C01734=2169.363,-41.196,-377.460,-0.2119,7.1275,-90.0002
C01735=2166.065,-41.196,-377.214,1.4381,5.5003,-90.0002
C01736=2165.275,-41.196,-377.323,0.1088,3.4320,-90.0002
C01737=2163.485,-41.196,-377.080,0.8193,6.3311,-90.0002
C01738=2160.102,-41.196,-377.738,1.1974,2.9163,-90.0002
C01739=2158.853,-41.196,-377.593,-1.1287,2.0683,-90.0002
C01740=2155.073,-41.196,-378.064,1.3693,1.9251,-90.0002
C01741=2153.724,-41.196,-377.850,1.3521,2.0282,-90.0002
C01742=2150.349,-41.196,-378.400,0.7620,2.9793,-90.0002
C01743=2149.136,-41.196,-377.910,3.1168,3.6783,-90.0002
C01744=2145.160,-41.196,-378.700,1.6558,3.1684,-90.0002
C01745=2144.326,-41.196,-378.466,1.6902,3.9190,-90.0002
C01746=2140.135,-41.196,-378.318,-1.0255,1.1459,-90.0002
C01747=2138.981,-41.196,-379.103,0.0114,2.0683,-90.0002
C01748=2135.291,-41.196,-378.850,3.2715,3.0710,-90.0002
C01749=2133.841,-41.196,-379.406,0.1718,0.1776,-90.0002
C01750=2130.488,-41.196,-378.890,4.1482,2.5840,-90.0002
C01751=2128.923,-41.196,-379.018,1.7990,7.3567,-90.0002
C01752=2125.737,-41.196,-379.393,3.4893,0.4526,-90.0002
C01753=2123.975,-41.196,-378.591,2.5954,1.8391,-90.0002
C01754=2120.075,-41.196,-379.170,-0.6073,2.3090,-90.0002
C01755=2118.901,-41.196,-379.712,0.9167,4.8185,-90.0002
C01756=2114.735,-41.196,-380.002,-3.3174,-0.1260,-90.0002
C01757=2113.577,-41.196,-379.959,2.9621,-3.2601,-90.0002
C01758=2110.098,-41.196,-379.433,10.2272,3.8674,-90.0002
C01759=2109.561,-41.196,-379.487,3.1971,-2.4293,-90.0002
C01760=2105.376,-41.196,-380.509,4.7440,3.5007,-90.0002
C01761=2104.898,-41.196,-379.374,1.4438,2.9679,-90.0002
C01762=2100.737,-41.196,-379.764,1.3521,-0.0458,-90.0002
C01763=2099.790,-41.196,-380.834,-1.4725,0.2291,-90.0002
C01764=2095.224,-41.196,-380.131,4.6123,2.7501,-90.0002
C01765=2093.930,-41.196,-380.331,1.6042,7.5859,-90.0002
C01766=2089.893,-41.196,-380.417,3.3976,4.7612,-90.0002
C01767=2089.258,-41.196,-380.773,0.7792,-1.9251,-90.0002
C01768=2085.330,-41.196,-380.757,0.7906,0.8193,-90.0002
C01769=2083.879,-41.196,-379.511,3.0194,-1.3980,-90.0002
C01770=2079.836,-41.196,-380.416,0.6245,0.3151,-90.0002
C01771=2079.038,-41.196,-380.368,2.0569,-1.8793,-90.0002
C01772=2074.672,-41.196,-379.861,3.7987,2.4980,-90.0002
C01773=2074.092,-41.196,-380.658,7.0473,8.2448,-90.0002
C01774=2070.056,-41.196,-379.715,-0.4640,3.1569,-90.0002
C01775=2069.076,-41.196,-380.400,-0.3265,-1.2776,-90.0002
C01776=2065.277,-41.196,-380.250,-0.5672,3.2773,-90.0002
C01777=2063.880,-41.196,-379.731,2.2517,-1.3808,-90.0002
C01778=2060.201,-41.196,-379.972,1.1631,-1.2318,-90.0002
C01779=2059.099,-41.196,-380.740,8.2276,1.3808,-90.0002
C01780=2055.123,-41.196,-380.849,3.2887,0.3495,-90.0002
C01781=2053.996,-41.196,-380.050,6.7551,-2.2230,-90.0002
C01782=2049.819,-41.196,-380.443,5.9358,-0.0687,-90.0002
C01783=2049.134,-41.196,-381.700,0.0229,5.6608,-90.0002
C01784=2045.224,-41.196,-381.245,5.5233,1.9595,-90.0002
C01785=2044.771,-41.196,-380.905,-4.0278,-0.0744,-90.0002
C01786=2040.257,-41.196,-381.458,1.0943,4.4633,-90.0002
C01787=2039.336,-41.196,-379.745,0.8880,1.7532,-90.0002
C01788=2035.560,-41.196,-380.149,0.7276,-3.2372,-90.0002
C01789=2033.515,-41.196,-381.337,1.0141,-2.7731,-90.0002
C01790=2029.970,-41.196,-381.111,4.8758,2.0912,-90.0002
C01791=2028.017,-41.196,-380.702,0.7505,-0.9052,-90.0002
C01792=2025.281,-41.196,-380.401,5.3800,-0.4297,-90.0002
C01793=2023.851,-41.196,-380.213,0.4812,-2.4350,-90.0002
C01794=2019.728,-41.196,-380.300,2.4121,-2.4006,-90.0002
C01795=2019.058,-41.196,-381.536,1.7647,2.5954,-90.0002
C01796=2014.946,-41.196,-380.978,1.1860,-0.4870,-90.0002
C01797=2010.390,-41.196,-380.567,-1.6386,5.3342,-90.0002
C01798=2009.731,-41.196,-381.456,3.9648,1.5068,-90.0002
C01799=2006.217,-41.196,-381.020,0.1546,3.9935,-90.0002
C01800=2004.385,-41.196,-380.094,1.2204,2.7903,-90.0002
C01801=2001.248,-41.196,-381.863,6.6692,5.0821,-90.0002
C01802=2000.379,-41.196,-380.943,5.5863,0.5500,-90.0002
C01803=1997.761,-41.196,-382.132,2.2116,-0.1718,-90.0002
C01804=1995.113,-41.196,-381.971,0.2578,3.1054,-90.0002
C01805=1994.652,-41.196,-379.974,2.1886,1.7074,-90.0002
C01806=1989.787,-41.196,-381.076,2.2173,-1.1229,-90.0002
C01807=1989.016,-41.196,-379.930,2.3491,0.3896,-90.0002
C01808=1986.291,-41.196,-381.148,-1.1688,-0.7047,-90.0002
C01809=1984.627,-41.196,-380.667,5.7467,2.3433,-90.0002
C01810=1980.711,-41.196,-381.395,3.0939,-0.4812,-90.0002
C01811=1980.047,-41.196,-381.569,2.0168,-4.2799,-90.0002
C01812=1976.640,-41.196,-382.374,6.9728,-1.3407,-90.0002
C01813=1975.100,-41.196,-380.121,-2.7845,0.1375,-90.0002
C01814=1973.698,-41.196,-381.294,-0.0802,5.6092,-90.0002
C01815=1970.010,-41.196,-380.203,9.3162,-2.5152,-90.0002
C01816=1968.613,-41.196,-382.095,-1.0313,1.8449,-90.0002
C01817=1966.022,-41.196,-381.592,3.9992,2.5439,-90.0002
C01818=1964.655,-41.196,-380.029,2.1314,1.8391,-90.0002
C01819=1960.547,-41.196,-380.255,2.1657,1.7188,-90.0002
C01820=1959.422,-41.196,-380.031,8.5198,-1.8678,-90.0002
C01821=1957.473,-41.196,-382.205,3.0997,-0.7792,-90.0002
C01822=1955.043,-41.196,-381.735,4.3945,0.1375,-90.0002
C01823=1954.062,-41.196,-381.684,6.5546,1.5412,-90.0002
C01824=1950.141,-41.196,-380.586,4.7956,0.8250,-90.0002
C01825=1949.476,-41.196,-381.977,1.8162,-8.2334,-90.0002
C01826=1945.507,-41.196,-381.667,1.2776,5.7926,-90.0002
C01827=1944.984,-41.196,-381.700,3.3861,2.4121,-90.0002
C01828=1943.695,-41.196,-382.237,-0.0114,2.3777,-90.0002
C01829=1941.079,-41.196,-381.081,1.8048,4.4633,-90.0002
C01830=1939.451,-41.196,-380.357,0.5385,3.7815,-90.0002
C01831=1935.406,-41.196,-381.487,2.2288,-1.6902,-90.0002
C01832=1934.176,-41.196,-380.632,5.7467,-0.7620,-90.0002
C01833=1930.488,-41.196,-381.185,6.1592,-2.4178,-90.0002
C01834=1929.880,-41.196,-381.659,-1.6844,0.4927,-90.0002
C01835=1926.074,-41.196,-380.394,0.8422,4.2112,-90.0002
C01836=1924.491,-41.196,-380.870,6.9728,-0.0974,-90.0002
C01837=1920.888,-41.196,-380.599,4.3201,4.1482,-90.0002
C01838=1920.372,-41.196,-381.287,7.0588,-6.8583,-90.0002
C01839=1919.171,-41.196,-382.295,0.0057,2.4465,-90.0002
C01840=1915.534,-41.196,-381.857,-6.9958,13.2295,-90.0002
C01841=1914.581,-41.196,-381.964,10.5137,-7.5401,-90.0002
C01842=1910.831,-41.196,-382.252,3.8846,-4.1825,-90.0002
C01843=1909.397,-41.196,-381.109,5.8040,0.4411,-90.0002
C01844=1905.433,-41.196,-381.982,5.2654,-2.9220,-90.0002
C01845=1904.354,-41.196,-380.850,4.1539,-1.1573,-90.0002
C01846=1901.224,-41.196,-380.146,1.1917,2.7845,-90.0002
C01847=1900.943,-41.196,-382.312,1.3407,-1.5813,-90.0002
C01848=1898.677,-41.196,-381.742,-0.9224,1.3235,-90.0002
C01849=1895.878,-41.196,-381.910,3.6096,-0.0630,-90.0002
C01850=1895.638,-41.196,-380.243,2.0397,1.5412,-90.0002
C01851=1892.807,-41.196,-382.261,0.9625,0.2005,-90.0002
C01852=1890.565,-41.196,-380.594,1.7074,1.1573,-90.0002
C01853=1889.860,-41.196,-381.233,-0.7964,-1.0599,-90.0002
C01854=1885.286,-41.196,-382.385,0.5786,1.4266,-90.0002
C01855=1884.612,-41.196,-380.791,1.2948,-0.9453,-90.0002
C01856=1882.779,-41.196,-382.009,3.6841,1.0370,-90.0002
C01857=1880.149,-41.196,-381.749,2.3720,-5.9301,-90.0002
C01858=1878.438,-41.196,-380.761,0.9511,-0.3609,-90.0002
C01859=1875.006,-41.196,-382.215,1.3063,-5.0935,-90.0002
C01860=1874.154,-41.196,-381.613,-1.0599,-0.8594,-90.0002
C01861=1870.916,-41.196,-381.373,1.7704,3.4893,-90.0002
C01862=1869.849,-41.196,-381.316,-0.6531,0.3896,-90.0002
C01863=1866.246,-41.196,-382.056,-1.6844,-6.2223,-90.0002
C01864=1864.858,-41.196,-379.990,2.8246,1.7761,-90.0002
C01865=1864.164,-41.196,-381.007,3.0022,0.7677,-90.0002
C01866=1859.806,-41.196,-380.511,1.6100,0.7677,-90.0002
C01867=1859.069,-41.196,-381.389,0.2521,-0.2922,-90.0002
C01868=1854.817,-41.196,-379.850,0.1489,4.6123,-90.0002
C01869=1853.868,-41.196,-381.034,5.8900,-1.4323,-90.0002
C01870=1850.003,-41.196,-380.905,2.6470,-0.5156,-90.0002
C01871=1848.676,-41.196,-380.548,0.7734,1.9938,-90.0002
C01872=1844.734,-41.196,-380.810,-1.4209,0.5958,-90.0002
C01873=1844.143,-41.196,-380.694,-1.6501,-0.9854,-90.0002
C01874=1840.047,-41.196,-379.707,4.4518,-5.9473,-90.0002
C01875=1838.314,-41.196,-379.343,1.3636,-3.0252,-90.0002
C01876=1834.393,-41.196,-379.620,-2.1084,0.3380,-90.0002
C01877=1833.918,-41.196,-380.668,2.2746,-6.1936,-90.0002
C01878=1829.774,-41.196,-379.832,-0.7448,-2.4522,-90.0002
C01879=1825.669,-41.196,-379.624,6.4973,-3.8903,-90.0002
C01880=1825.187,-41.196,-379.253,3.0825,-5.2368,-90.0002
C01881=1820.708,-41.196,-378.938,2.6871,-3.0137,-90.0002
C01882=1819.044,-41.196,-379.962,-0.4469,1.3120,-90.0002
C01883=1815.594,-41.196,-379.344,3.0194,-0.9224,-90.0002
C01884=1814.615,-41.196,-378.950,3.4320,-2.8132,-90.0002
C01885=1810.688,-41.196,-379.312,-0.1661,-2.1027,-90.0002
C01886=1809.855,-41.196,-379.145,4.2857,-2.7673,-90.0002
C01887=1805.671,-41.196,-378.925,0.2922,-3.3747,-90.0002
C01888=1804.704,-41.196,-378.996,2.3605,-4.5492,-90.0002
C01889=1800.366,-41.196,-378.306,4.3201,-5.8327,-90.0002
C01890=1799.418,-41.196,-378.526,-5.2941,-12.6394,-90.0002
C01891=1795.305,-91.196,-377.541,1.0542,7.1104,-90.0002
C01892=1799.418,-91.196,-377.424,1.8162,-5.2712,-90.0002
C01893=1800.080,-91.196,-377.530,-0.8995,-6.1134,-90.0002
C01894=1804.178,-91.196,-377.422,0.5271,-1.1631,-90.0002
C01895=1805.558,-91.196,-378.041,2.7272,-4.0794,-90.0002
C01896=1809.552,-91.196,-378.343,-0.9224,3.0997,-90.0002
C01897=1810.802,-91.196,-377.922,2.2803,-1.4037,-90.0002
C01898=1814.674,-91.196,-377.946,-0.2177,2.1543,-90.0002
C01899=1816.221,-91.196,-377.447,4.0278,1.1401,-90.0002
C01900=1819.459,-91.196,-378.316,0.6245,-1.4495,-90.0002
C01901=1820.188,-91.196,-378.633,3.9190,-3.7757,-90.0002
C01902=1823.981,-91.196,-378.201,0.4984,0.5786,-90.0002
C01903=1825.225,-91.196,-377.414,3.6039,0.5729,-90.0002
C01904=1829.473,-91.196,-377.953,3.6898,0.2119,-90.0002
C01905=1830.985,-91.196,-378.696,-0.7906,0.8307,-90.0002
C01906=1834.377,-91.196,-377.651,1.8506,3.2544,-90.0002
C01907=1835.959,-91.196,-377.260,0.4640,-0.9568,-90.0002
C01908=1839.694,-91.196,-377.295,2.4923,-0.5213,-90.0002
C01909=1840.541,-91.196,-378.454,2.9507,-6.2395,-90.0002
C01910=1844.696,-91.196,-377.160,0.1948,2.4064,-90.0002
C01911=1845.955,-91.196,-377.972,3.5809,-0.0744,-90.0002
C01912=1848.927,-91.196,-378.948,6.5145,-2.1428,-90.0002
C01913=1849.965,-91.196,-377.457,4.4518,1.1516,-90.0002
C01914=1851.787,-91.196,-376.910,4.3258,-2.3949,-90.0002
C01915=1854.842,-91.196,-377.542,1.1401,2.7501,-90.0002
C01916=1855.268,-91.196,-378.573,2.6699,-0.3781,-90.0002
C01917=1859.702,-91.196,-378.097,3.0481,0.3781,-90.0002
C01918=1860.339,-91.196,-377.126,1.4839,4.8930,-90.0002
C01919=1864.837,-91.196,-377.522,2.1600,-1.5870,-90.0002
C01920=1866.502,-91.196,-378.692,-1.9938,1.4323,-90.0002
C01921=1869.655,-91.196,-379.088,5.2712,0.2807,-90.0002
C01922=1870.902,-91.196,-378.347,3.7929,3.7471,-90.0002
C01923=1874.608,-91.196,-378.370,7.1275,-2.7215,-90.0002
C01924=1875.701,-91.196,-377.271,2.4694,1.8964,-90.0002
C01925=1879.089,-91.196,-376.878,2.4522,0.1890,-90.0002
C01926=1880.404,-91.196,-377.206,2.2918,-0.0229,-90.0002
C01927=1883.226,-91.196,-379.326,1.9767,-3.0366,-90.0002
C01928=1884.972,-91.196,-378.617,0.3953,1.4094,-90.0002
C01929=1889.337,-91.196,-377.344,5.2597,-0.7391,-90.0002
C01930=1890.538,-91.196,-377.879,3.6726,0.8880,-90.0002
C01931=1894.036,-91.196,-376.879,1.2948,2.3605,-90.0002
C01932=1895.783,-91.196,-378.730,7.9984,-2.5496,-90.0002
C01933=1899.291,-91.196,-379.024,3.5179,0.5156,-90.0002
C01934=1900.259,-91.196,-378.071,3.0022,-0.2807,-90.0002
C01935=1902.386,-91.196,-377.434,4.2341,-4.2742,-90.0002
C01936=1905.020,-91.196,-378.297,11.6596,4.2055,-90.0002
C01937=1907.374,-91.196,-379.871,1.9652,2.2459,-90.0002
C01938=1909.572,-91.196,-377.869,1.4839,1.8964,-90.0002
C01939=1910.710,-91.196,-377.032,4.0508,-1.7589,-90.0002
C01940=1914.960,-91.196,-379.427,4.7841,0.5786,-90.0002
C01941=1915.743,-91.196,-378.526,1.3235,-1.5297,-90.0002
C01942=1920.119,-91.196,-379.065,4.4919,1.5297,-90.0002
C01943=1920.959,-91.196,-378.296,-0.0229,4.7612,-90.0002
C01944=1924.741,-91.196,-380.206,2.2402,0.7563,-90.0002
C01945=1925.292,-91.196,-378.183,2.6757,-5.1050,-90.0002
C01946=1930.023,-91.196,-377.070,6.5202,3.2715,-90.0002
C01947=1930.189,-91.196,-378.390,5.8842,1.1287,-90.0002
C01948=1934.079,-91.196,-376.687,-2.3835,0.8365,-90.0002
C01949=1935.446,-91.196,-379.999,3.5065,1.0828,-90.0002
C01950=1938.838,-91.196,-377.816,2.6356,-0.9682,-90.0002
C01951=1940.436,-91.196,-378.391,4.4346,1.6157,-90.0002
C01952=1942.886,-91.196,-379.959,0.6932,2.2116,-90.0002
C01953=1944.917,-91.196,-377.943,4.2799,1.9365,-90.0002
C01954=1948.261,-91.196,-377.396,3.0595,1.5469,-90.0002
C01955=1949.956,-91.196,-378.329,1.3349,0.4984,-90.0002
C01956=1953.464,-91.196,-377.372,3.5179,-1.6730,-90.0002
C01957=1955.037,-91.196,-379.269,1.9365,2.7960,-90.0002
C01958=1957.644,-91.196,-377.607,1.7475,2.2689,-90.0002
C01959=1959.560,-91.196,-379.741,2.5783,7.5802,-90.0002
C01960=1963.395,-91.196,-378.215,7.7463,0.4411,-90.0002
C01961=1964.946,-91.196,-376.641,3.7643,-0.8537,-90.0002
C01962=1969.099,-91.196,-378.729,5.1050,1.8506,-90.0002
C01963=1970.306,-91.196,-377.055,3.7414,-0.1833,-90.0002
C01964=1972.157,-91.196,-376.780,0.7792,1.5584,-90.0002
C01965=1974.946,-91.196,-378.646,2.7158,-0.2692,-90.0002
C01966=1975.717,-91.196,-379.977,7.0359,0.8766,-90.0002
C01967=1979.866,-91.196,-378.788,-0.4755,-0.8250,-90.0002
C01968=1981.044,-91.196,-377.480,2.2918,0.4640,-90.0002
C01969=1984.927,-91.196,-379.068,4.5607,0.6589,-90.0002
C01970=1987.335,-91.196,-376.378,4.2055,2.3491,-90.0002
C01971=1990.373,-91.196,-378.245,3.0080,1.4266,-90.0002
C01972=1992.305,-91.196,-379.490,2.4236,0.7964,-90.0002
C01973=1994.371,-91.196,-379.740,6.0790,0.5500,-90.0002
C01974=1995.503,-91.196,-379.443,0.4927,-1.7761,-90.0002
C01975=1999.561,-91.196,-377.473,1.5183,2.2173,-90.0002
C01976=2000.080,-91.196,-379.228,1.2891,2.9621,-90.0002
C01977=2004.406,-91.196,-378.900,-1.6501,2.0683,-90.0002
C01978=2005.652,-91.196,-377.941,2.6184,0.8021,-90.0002
C01979=2009.434,-91.196,-378.794,0.4239,-3.4492,-90.0002
C01980=2010.261,-91.196,-377.289,2.8361,-0.6245,-90.0002
C01981=2013.853,-91.196,-379.442,2.9621,4.2112,-90.0002
C01982=2015.071,-91.196,-377.219,2.6585,2.2402,-90.0002
C01983=2019.320,-91.196,-379.177,3.7815,-0.5844,-90.0002
C01984=2020.278,-91.196,-377.598,4.4919,3.1226,-90.0002
C01985=2024.061,-91.196,-378.312,1.9365,2.6012,-90.0002
C01986=2024.673,-91.196,-377.500,5.7467,1.0485,-90.0002
C01987=2028.765,-91.196,-377.287,3.8388,-5.4717,-90.0002
C01988=2029.403,-91.196,-379.302,-2.2345,-1.3063,-90.0002
C01989=2033.995,-91.196,-379.271,2.9278,1.7246,-90.0002
C01990=2035.196,-91.196,-377.121,4.8185,0.4526,-90.0002
C01991=2036.257,-91.196,-376.721,10.1528,2.3720,-90.0002
C01992=2040.109,-91.196,-378.754,7.9354,0.5500,-90.0002
C01993=2041.225,-91.196,-377.911,-0.4411,1.0657,-90.0002
C01994=2044.180,-91.196,-379.373,2.9335,-1.6386,-90.0002
C01995=2044.990,-91.196,-377.271,1.3521,4.0164,-90.0002
C01996=2049.316,-91.196,-379.066,6.3025,-1.2662,-90.0002
C01997=2050.431,-91.196,-379.407,0.5786,1.3865,-90.0002
C01998=2054.812,-91.196,-378.624,0.2234,0.9625,-90.0002
C01999=2055.478,-91.196,-377.232,6.3999,-2.6356,-90.0002
C02000=2059.087,-91.196,-379.472,4.1825,1.1229,-90.0002
C02001=2060.348,-91.196,-379.251,4.4862,4.9045,-90.0002
C02002=2064.525,-91.196,-377.693,3.4320,0.2521,-90.0002
C02003=2065.787,-91.196,-377.027,1.9308,-1.4725,-90.0002
C02004=2067.675,-91.196,-377.871,5.0305,-0.0630,-90.0002
C02005=2069.595,-91.196,-376.894,2.4694,1.2433,-90.0002
C02006=2070.674,-91.196,-378.584,6.5947,2.0053,-90.0002
C02007=2074.375,-91.196,-378.345,4.0393,-0.8021,-90.0002
C02008=2075.996,-91.196,-378.574,2.9564,-0.6359,-90.0002
C02009=2079.628,-91.196,-379.307,-2.1314,-1.5183,-90.0002
C02010=2080.836,-91.196,-378.302,5.6837,1.9079,-90.0002
C02011=2084.764,-91.196,-378.169,-0.6932,0.1145,-90.0002
C02012=2086.437,-91.196,-376.636,5.5977,-1.2032,-90.0002
C02013=2089.410,-91.196,-378.030,0.8766,3.1569,-90.0002
C02014=2090.183,-91.196,-377.411,2.8647,3.1111,-90.0002
C02015=2094.448,-91.196,-378.114,2.3032,-0.5901,-90.0002
C02016=2096.058,-91.196,-377.332,1.9767,2.8590,-90.0002
C02017=2099.543,-91.196,-377.890,6.0160,0.3380,-90.0002
C02018=2100.315,-91.196,-378.222,3.9534,-0.4297,-90.0002
C02019=2104.184,-91.196,-376.632,5.2024,-2.3777,-90.0002
C02020=2104.790,-91.196,-377.159,2.6642,0.0802,-90.0002
C02021=2107.833,-91.196,-376.917,4.3544,1.6673,-90.0002
C02022=2110.286,-91.196,-378.242,5.9301,1.0599,-90.0002
C02023=2111.691,-91.196,-377.226,4.3659,6.2108,-90.0002
C02024=2114.634,-91.196,-378.486,0.7964,-1.5527,-90.0002
C02025=2116.213,-91.196,-378.735,6.7150,2.4579,-90.0002
C02026=2119.530,-91.196,-376.715,0.9453,-0.0572,-90.0002
C02027=2121.044,-91.196,-377.621,1.9136,2.3090,-90.0002
C02028=2124.313,-91.196,-377.459,4.4633,4.2456,-90.0002
C02029=2125.062,-91.196,-377.243,4.1711,-1.2891,-90.0002
C02030=2128.421,-91.196,-376.976,5.2425,3.3575,-90.0002
C02031=2129.559,-91.196,-377.491,1.8277,3.9476,-90.0002
C02032=2131.041,-91.196,-378.289,2.2975,4.6581,-90.0002
C02033=2134.586,-91.196,-377.315,2.7731,2.5095,-90.0002
C02034=2135.602,-91.196,-377.583,1.8162,2.5382,-90.0002
C02035=2138.526,-91.196,-377.954,1.0084,4.3029,-90.0002
C02036=2140.068,-91.196,-376.562,2.3032,4.4919,-90.0002
C02037=2141.212,-91.196,-376.416,1.2032,6.1478,-90.0002
C02038=2144.686,-91.196,-376.860,0.7448,1.8964,-90.0002
C02039=2145.499,-91.196,-376.622,1.1344,0.4239,-90.0002
C02040=2149.245,-91.196,-377.512,3.1512,1.4209,-90.0002
C02041=2150.530,-91.196,-376.290,2.6871,1.9652,-90.0002
C02042=2154.261,-91.196,-375.625,1.7818,4.1711,-90.0002
C02043=2155.389,-91.196,-377.406,-0.5328,5.5003,-90.0002
C02044=2158.923,-91.196,-376.796,3.0424,2.1027,-90.0002
C02045=2159.995,-91.196,-377.108,2.1886,5.3800,-90.0002
C02046=2162.658,-91.196,-377.093,-2.9278,1.2776,-90.0002
C02047=2165.115,-91.196,-376.774,-1.1459,1.9767,-90.0002
C02048=2166.465,-91.196,-376.259,1.1344,0.3208,-90.0002
C02049=2169.854,-91.196,-376.573,2.2631,3.6096,-90.0002
C02050=2171.046,-91.196,-376.056,-0.4526,0.4812,-90.0002
C02051=2174.160,-91.196,-376.291,4.0278,3.7987,-90.0002
C02052=2175.265,-91.196,-375.729,4.2398,3.4434,-90.0002
C02053=2179.561,-91.196,-375.441,-1.2948,4.6810,-90.0002
C02054=2180.555,-91.196,-376.351,3.7184,6.6978,-90.0002
C02055=2184.038,-91.196,-375.049,-0.9453,5.4201,-90.0002
C02056=2185.498,-91.196,-374.824,6.5374,3.6268,-90.0002
C02057=2185.415,-141.196,-374.060,2.6699,2.4178,-90.0002
C02058=2184.214,-141.196,-373.905,3.8388,-0.5328,-90.0002
C02059=2180.012,-141.196,-374.573,-0.2750,1.7188,-90.0002
C02060=2179.127,-141.196,-373.260,4.8414,1.6558,-90.0002
C02061=2175.684,-141.196,-373.842,2.8074,1.6157,-90.0002
C02062=2174.219,-141.196,-375.290,0.1203,1.9938,-90.0002
C02063=2170.489,-141.196,-374.723,0.7505,-0.1432,-90.0002
C02064=2169.134,-141.196,-375.269,2.4465,0.8823,-90.0002
C02065=2165.315,-141.196,-373.747,5.3399,2.9450,-90.0002
C02066=2164.630,-141.196,-375.232,1.5928,-2.0511,-90.0002
C02067=2160.260,-141.196,-374.253,3.2486,-0.4755,-90.0002
C02068=2159.387,-141.196,-375.240,3.2085,2.3204,-90.0002
C02069=2155.362,-141.196,-374.889,3.2601,2.3376,-90.0002
C02070=2154.922,-141.196,-375.396,1.6443,-3.1054,-90.0002
C02071=2150.433,-141.196,-374.026,6.6119,0.3208,-90.0002
C02072=2149.135,-141.196,-374.393,2.4350,0.5901,-90.0002
C02073=2145.477,-141.196,-375.714,3.7356,1.0370,-90.0002
C02074=2144.146,-141.196,-373.491,9.5512,2.5897,-90.0002
C02075=2140.769,-141.196,-374.776,5.0248,-0.2922,-90.0002
C02076=2139.289,-141.196,-373.542,7.4140,-1.3922,-90.0002
C02077=2135.263,-141.196,-375.429,7.3510,0.1833,-90.0002
C02078=2133.968,-141.196,-373.056,1.0886,0.0744,-90.0002
C02079=2130.077,-141.196,-375.677,3.5408,2.3204,-90.0002
C02080=2129.113,-141.196,-373.373,6.1077,-0.3609,-90.0002
C02081=2125.272,-141.196,-375.578,2.2345,-0.4755,-90.0002
C02082=2124.761,-141.196,-376.048,2.3835,1.5240,-90.0002
C02083=2120.328,-141.196,-375.059,4.2799,3.1856,-90.0002
C02084=2118.606,-141.196,-375.500,2.9048,-1.3407,-90.0002
C02085=2115.318,-141.196,-372.750,6.7666,5.3055,-90.0002
C02086=2113.745,-141.196,-375.727,1.9423,2.2116,-90.0002
C02087=2110.355,-141.196,-376.311,2.8762,2.6642,-90.0002
C02088=2109.416,-141.196,-375.774,2.6757,1.2146,-90.0002
C02089=2105.001,-141.196,-375.638,5.5061,-0.5557,-90.0002
C02090=2104.265,-141.196,-372.948,9.5397,-1.5412,-90.0002
C02091=2100.516,-141.196,-375.890,3.7815,0.3208,-90.0002
C02092=2099.725,-141.196,-375.017,5.3514,2.5954,-90.0002
C02093=2095.436,-141.196,-374.505,3.1340,-2.1886,-90.0002
C02094=2094.167,-141.196,-374.712,7.3968,-1.4725,-90.0002
C02095=2090.205,-141.196,-375.986,1.2204,-0.8938,-90.0002
C02096=2089.109,-141.196,-374.205,4.1310,-2.1715,-90.0002
C02097=2085.580,-141.196,-375.997,3.4148,-0.6703,-90.0002
C02098=2084.360,-141.196,-374.346,4.7727,-0.3495,-90.0002
C02099=2080.253,-141.196,-373.722,6.0160,1.6902,-90.0002
C02100=2079.835,-141.196,-376.286,5.4602,1.1000,-90.0002
C02101=2074.913,-141.196,-376.787,5.9702,-1.1172,-90.0002
C02102=2073.522,-141.196,-375.699,5.3055,-0.2922,-90.0002
C02103=2069.173,-141.196,-373.234,4.2226,0.9281,-90.0002
C02104=2066.401,-141.196,-374.355,0.6760,1.9365,-90.0002
C02105=2064.927,-141.196,-375.525,1.1631,1.4495,-90.0002
C02106=2061.460,-141.196,-375.886,-0.9912,3.4033,-90.0002
C02107=2059.609,-141.196,-376.501,3.9648,-1.4495,-90.0002
C02108=2055.666,-141.196,-376.502,3.8903,0.3380,-90.0002
C02109=2055.045,-141.196,-375.888,1.5641,-0.8307,-90.0002
C02110=2051.232,-141.196,-374.111,-0.0171,1.5297,-90.0002
C02111=2049.797,-141.196,-376.208,7.0989,1.1287,-90.0002
C02112=2046.719,-141.196,-376.168,5.1508,1.7131,-90.0002
C02113=2045.239,-141.196,-372.335,-0.4927,-0.3609,-90.0002
C02114=2041.406,-141.196,-374.903,1.2433,1.2032,-90.0002
C02115=2039.762,-141.196,-374.660,3.5007,0.2291,-90.0002
C02116=2036.008,-141.196,-373.939,10.2158,2.8017,-90.0002
C02117=2034.926,-141.196,-373.407,8.3823,-1.5756,-90.0002
C02118=2030.385,-141.196,-374.996,4.5951,-1.0198,-90.0002
C02119=2029.826,-141.196,-374.272,9.8319,-2.3204,-90.0002
C02120=2026.054,-141.196,-375.886,3.5351,0.4812,-90.0002
C02121=2024.793,-141.196,-372.708,0.9339,2.4236,-90.0002
C02122=2020.791,-141.196,-373.674,11.6997,-2.9450,-90.0002
C02123=2019.172,-141.196,-375.199,3.9133,-0.1948,-90.0002
C02124=2016.262,-141.196,-377.076,2.7845,5.8728,-90.0002
C02125=2014.369,-141.196,-375.197,2.3720,0.4239,-90.0002
C02126=2010.352,-141.196,-374.971,4.6810,0.2864,-90.0002
C02127=2009.288,-141.196,-376.093,6.0504,0.8594,-90.0002
C02128=2005.597,-141.196,-375.731,5.6780,0.0802,-90.0002
C02129=2004.514,-141.196,-376.381,6.5890,-0.5786,-90.0002
C02130=2000.011,-141.196,-373.316,8.7719,4.5034,-90.0002
C02131=1998.643,-141.196,-376.369,3.5637,-1.1229,-90.0002
C02132=1995.495,-141.196,-375.756,6.1478,4.0966,-90.0002
C02133=1994.531,-141.196,-374.155,9.4251,-1.5011,-90.0002
C02134=1990.070,-141.196,-375.098,3.0653,-0.6646,-90.0002
C02135=1989.589,-141.196,-374.441,5.6608,3.1111,-90.0002
C02136=1984.910,-141.196,-374.777,0.8078,4.3716,-90.0002
C02137=1983.861,-141.196,-374.952,4.2971,3.1398,-90.0002
C02138=1980.391,-141.196,-374.252,6.0561,0.0744,-90.0002
C02139=1979.309,-141.196,-375.340,3.8617,1.5641,-90.0002
C02140=1975.109,-141.196,-376.260,6.2051,1.6214,-90.0002
C02141=1974.206,-141.196,-375.762,3.0538,0.6302,-90.0002
C02142=1970.228,-141.196,-374.936,2.1428,1.0599,-90.0002
C02143=1969.207,-141.196,-375.892,6.8697,0.3265,-90.0002
C02144=1965.515,-141.196,-375.103,3.5924,-0.9682,-90.0002
C02145=1964.102,-141.196,-376.394,5.5691,-2.4809,-90.0002
C02146=1959.717,-141.196,-375.815,4.2513,-0.8537,-90.0002
C02147=1959.054,-141.196,-373.895,3.7184,3.0767,-90.0002
C02148=1954.785,-141.196,-374.983,3.5236,0.0859,-90.0002
C02149=1954.384,-141.196,-375.969,-0.4239,3.3632,-97.1679
C02150=1950.054,-141.196,-375.487,2.4293,0.0458,-90.0002
C02151=1949.440,-141.196,-375.245,4.0565,-0.9110,-90.0002
C02152=1945.526,-141.196,-376.724,4.3602,-2.4522,-90.0002
C02153=1944.222,-141.196,-374.130,9.6027,-4.0107,-90.0002
C02154=1940.229,-141.196,-376.375,5.8842,1.6902,-90.0002
C02155=1939.527,-141.196,-377.085,-0.1088,1.1287,-90.0002
C02156=1935.213,-141.196,-373.944,3.5867,-1.9652,-90.0002
C02157=1934.819,-141.196,-375.337,5.0133,1.1058,-90.0002
C02158=1930.636,-141.196,-375.890,2.6012,0.0401,-90.0002
C02159=1929.735,-141.196,-376.410,1.7360,0.2005,-90.0002
C02160=1925.900,-141.196,-375.823,4.8987,-0.6646,-90.0002
C02161=1924.700,-141.196,-373.832,4.6696,-0.6818,-90.0002
C02162=1920.470,-141.196,-376.522,1.8964,1.4839,-90.0002
C02163=1919.832,-141.196,-376.398,7.0588,-1.1631,-90.0002
C02164=1916.892,-141.196,-375.801,5.0305,0.0802,-90.0002
C02165=1915.052,-141.196,-373.246,1.3750,1.9423,-90.0002
C02166=1912.060,-141.196,-376.956,4.9790,-0.6302,-90.0002
C02167=1910.298,-141.196,-375.968,2.0511,1.5412,-90.0002
C02168=1908.582,-141.196,-376.159,2.2975,3.9190,-90.0002
C02169=1905.388,-141.196,-373.909,6.9098,-4.0336,-90.0002
C02170=1903.985,-141.196,-376.680,3.2314,-0.8250,-90.0002
C02171=1900.049,-141.196,-376.768,-0.3093,0.4068,-90.0002
C02172=1899.194,-141.196,-376.566,4.7383,2.8819,-90.0002
C02173=1895.499,-141.196,-374.703,3.2715,2.5954,-90.0002
C02174=1894.268,-141.196,-376.976,1.5240,-1.5355,-90.0002
C02175=1890.500,-141.196,-375.186,9.5913,3.0080,-90.0002
C02176=1889.495,-141.196,-376.046,3.0080,0.1031,-90.0002
C02177=1885.342,-141.196,-376.640,3.3976,-0.3495,-90.0002
C02178=1885.135,-141.196,-375.791,3.1512,-0.9167,-90.0002
C02179=1879.748,-141.196,-375.833,6.2509,-0.8880,-90.0002
C02180=1878.976,-141.196,-375.179,7.6088,-2.4236,-90.0002
C02181=1875.506,-141.196,-376.619,9.7116,-2.7330,-90.0002
C02182=1874.493,-141.196,-374.949,6.0504,0.3609,-90.0002
C02183=1870.194,-141.196,-374.646,5.2540,3.8617,-90.0002
C02184=1869.293,-141.196,-375.463,3.0366,-0.4984,-90.0002
C02185=1865.075,-141.196,-376.316,2.4064,1.6787,-90.0002
C02186=1864.404,-141.196,-375.624,0.4125,2.3376,-90.0002
C02187=1859.803,-141.196,-375.872,2.1715,0.4927,-90.0002
C02188=1858.398,-141.196,-375.605,3.1340,-0.1432,-90.0002
C02189=1854.864,-141.196,-375.996,3.0767,-0.0859,-90.0002
C02190=1853.834,-141.196,-374.837,2.2918,1.4266,-90.0002
C02191=1850.410,-141.196,-375.284,2.2746,3.0080,-90.0002
C02192=1849.748,-141.196,-375.547,2.7501,1.1172,-90.0002
C02193=1845.055,-141.196,-375.674,3.4090,5.7123,-90.0002
C02194=1844.434,-141.196,-377.106,-3.7643,7.5401,-90.0002
C02195=1840.894,-141.196,-375.702,1.3063,-0.7333,-90.0002
C02196=1839.805,-141.196,-376.567,1.8621,1.5813,-90.0002
C02197=1835.935,-141.196,-377.111,1.0198,-2.9908,-90.0002
C02198=1834.687,-141.196,-375.834,8.2964,1.2547,-90.0002
C02199=1832.895,-141.196,-376.758,1.9022,-0.5213,-90.0002
C02200=1829.331,-141.196,-375.944,13.2410,2.8304,-90.0002
C02201=1825.616,-141.196,-376.772,2.5496,-2.2975,-90.0002
C02202=1824.719,-141.196,-376.707,-0.7161,2.4236,-90.0002
C02203=1823.375,-141.196,-376.275,1.4610,2.5954,-90.0002
C02204=1820.148,-141.196,-376.699,0.9224,1.9022,-90.0002
C02205=1819.386,-141.196,-377.239,-0.7333,7.9411,-90.0002
C02206=1817.633,-141.196,-377.017,-4.0794,7.6203,-90.0002
C02207=1815.194,-141.196,-377.208,0.9224,0.3208,-90.0002
C02208=1813.793,-141.196,-377.163,2.0741,-0.5271,-90.0002
C02209=1810.514,-141.196,-376.879,1.0370,0.4583,-90.0002
C02210=1809.304,-141.196,-376.514,5.6035,5.9358,-90.0002
C02211=1805.917,-141.196,-377.286,1.4438,1.7016,-90.0002
C02212=1805.150,-141.196,-377.071,-1.3120,3.1398,-90.0002
C02213=1803.613,-141.196,-376.936,4.8357,-1.0198,-90.0002
C02214=1800.646,-141.196,-376.815,1.7417,1.7475,-90.0002
C02215=1799.896,-141.196,-377.079,-1.0026,0.1203,-90.0002
C02216=1798.042,-141.196,-377.026,0.1088,5.4488,-90.0002
C02217=1794.253,-141.196,-377.324,1.7188,11.2528,-90.0002
C02218=1812.109,341.105,-503.612,89.8111,-0.2349,0.0000
C02219=2127.650,341.132,-503.612,90.5788,-0.2750,0.0000
C02220=2159.023,341.159,-503.612,90.6075,-0.4927,-0.0057
C02221=1816.234,341.190,-503.612,89.6048,0.1546,0.0000
C02222=1821.738,341.222,-503.612,90.0002,0.0687,0.0000
C02223=1812.786,341.237,-503.612,89.4559,-0.2922,0.0000
C02224=1809.568,341.249,-503.612,83.1648,0.5213,-0.0630
C02225=1831.712,341.267,-503.612,89.6621,0.4927,-0.0057
C02226=1826.384,341.287,-503.612,89.5475,0.2119,0.0000
C02227=1835.441,341.299,-503.612,89.7309,0.1145,0.0000
C02228=1840.177,341.323,-503.612,89.6736,0.4583,0.0000
C02229=1835.884,341.334,-503.612,89.8798,0.2406,0.0000
C02230=2119.313,341.341,-503.612,89.6335,0.1489,0.0000
C02231=2152.042,341.346,-503.612,90.8309,0.0229,0.0000
C02232=2175.237,341.354,-503.612,90.0403,0.4068,0.0000
C02233=1808.484,341.385,-503.612,89.6163,-1.0026,0.0057
C02234=2144.675,341.398,-503.612,90.8596,-0.2807,-0.0057
C02235=1798.586,341.407,-503.612,89.6392,0.8365,-0.0057
C02236=1838.296,341.417,-503.612,89.5361,-0.7677,0.0057
C02237=2112.907,341.440,-503.612,90.9513,-0.7849,-0.0114
C02238=2136.688,341.448,-503.612,90.9627,-0.2750,-0.0057
C02239=2090.048,341.463,-503.612,91.0258,-0.1661,-0.0057
C02240=1866.740,341.476,-503.612,84.0930,-0.0343,0.0057
C02241=2119.757,341.491,-503.612,90.7565,-0.3552,-0.0057
C02242=1858.245,341.509,-503.612,90.4528,0.4583,0.0057
C02243=2166.766,341.523,-503.612,90.9398,0.5385,0.0114
C02244=1851.449,341.538,-503.612,90.6705,0.8422,0.0114
C02245=2144.147,341.553,-503.612,90.6018,-0.2291,0.0000
C02246=1829.104,341.580,-503.612,86.4765,0.5328,-0.0343
C02247=1861.433,341.584,-503.612,89.6392,0.4469,0.0000
C02248=2184.909,341.594,-503.612,89.5819,1.9136,-0.0114
C02249=2091.279,341.606,-503.612,90.9914,-1.0026,-0.0171
C02250=1817.924,341.619,-503.612,88.7511,4.3086,-0.0916
C02251=2128.544,341.634,-503.612,75.2580,0.4010,-0.1031
C02252=2189.650,341.644,-503.612,91.6789,-4.6065,-0.1375
C02253=2117.508,341.652,-503.612,90.4127,-0.3093,0.0000
C02254=2109.284,341.657,-503.612,89.6507,-0.7219,0.0057
C02255=2090.436,341.673,-503.612,91.8795,0.0343,0.0000
C02256=2114.097,341.679,-503.612,90.2695,-0.2119,0.0000
C02257=2126.105,341.684,-503.612,91.1919,0.4125,0.0114
C02258=2089.212,341.696,-503.612,89.7996,-0.5614,0.0000
C02259=1866.067,341.706,-503.612,89.8970,0.8708,0.0000
C02260=2127.724,341.717,-503.612,90.7679,0.1375,0.0000
C02261=2081.920,341.730,-503.612,90.7335,-1.1459,-0.0171
C02262=2079.389,341.738,-503.612,90.0288,-0.4526,0.0000
C02263=1876.495,341.751,-503.612,89.4215,1.0255,-0.0114
C02264=1875.989,341.764,-503.612,77.3550,0.4469,-0.1031
C02265=2183.623,341.792,-503.612,90.5846,1.7016,0.0171
C02266=2072.497,341.803,-503.612,90.2064,-0.4010,0.0000
C02267=2080.170,341.818,-503.612,90.4127,-0.4182,-0.0057
C02268=1887.562,341.829,-503.612,90.0804,1.0026,0.0000
C02269=2189.014,341.847,-503.612,89.7939,-3.8731,0.0114
C02270=2076.462,341.853,-503.612,89.5934,-0.6760,0.0057
C02271=2063.601,341.860,-503.612,89.9257,-0.5844,0.0000
C02272=1880.479,341.880,-503.612,90.0116,1.1745,0.0000
C02273=2072.651,341.889,-503.612,90.3267,-0.1833,0.0000
C02274=2142.630,341.920,-503.612,91.4383,0.6417,0.0171
C02275=2163.746,341.939,-503.612,82.6205,0.8880,-0.1145
C02276=2043.757,341.950,-503.612,90.0288,0.2119,0.0000
C02277=2143.560,341.978,-503.612,80.5922,0.4182,-0.0687
C02278=2152.254,341.994,-503.612,86.4077,-0.9912,0.0630
C02279=1890.422,342.008,-503.612,89.2324,0.8880,-0.0114
C02280=2187.978,342.021,-503.612,93.6442,-0.2406,-0.0171
C02281=1997.694,342.034,-503.612,88.8371,-8.1761,0.1661
C02282=1909.060,342.052,-503.612,90.8539,1.0828,0.0171
C02283=1902.578,342.072,-503.612,89.7423,0.6417,-0.0057
C02284=1894.728,342.089,-503.612,90.1377,1.3750,0.0057
C02285=2088.376,342.092,-503.612,86.3676,-2.0454,0.1317
C02286=1919.373,342.116,-503.612,88.9631,1.2719,-0.0229
C02287=1998.261,342.133,-503.612,87.5364,-1.9824,0.0859
C02288=1997.057,342.151,-503.612,89.0261,-0.3323,0.0057
C02289=1985.819,342.166,-503.612,83.3596,2.4637,-0.2864
C02290=1910.512,342.177,-503.612,81.8355,0.2291,-0.0343
C02291=2049.023,342.193,-503.612,90.5330,-0.0458,0.0000
C02292=2036.066,342.204,-503.612,90.2351,-0.5557,0.0000
C02293=2032.569,342.235,-503.612,89.7481,-0.2406,0.0000
C02294=1901.945,342.245,-503.612,89.4960,1.0485,-0.0114
C02295=1912.115,342.262,-503.612,89.1293,1.2776,-0.0171
C02296=2025.810,342.269,-503.612,89.6048,0.0744,0.0000
C02297=1898.412,342.295,-503.612,86.4765,-0.8479,0.0515
C02298=2029.161,342.309,-503.612,85.6629,-0.3437,0.0286
C02299=1902.070,342.318,-503.612,90.1205,1.8277,0.0057
C02300=1927.560,342.328,-503.612,88.9287,0.5614,-0.0114
C02301=2003.102,342.352,-503.612,89.2610,-0.1776,0.0000
C02302=1982.107,342.368,-503.612,90.2122,-0.5672,0.0000
C02303=2008.875,342.379,-503.612,89.3069,0.0859,0.0000
C02304=2017.438,342.392,-503.612,89.4387,-0.2463,0.0000
C02305=1928.227,342.404,-503.612,83.8351,-0.0859,0.0114
C02306=1937.098,342.419,-503.612,88.6995,-0.5271,0.0114
C02307=1942.371,342.434,-503.612,88.4131,-0.0057,0.0000
C02308=1916.394,342.451,-503.612,89.7481,0.5557,0.0000
C02309=1942.013,342.472,-503.612,89.4501,0.2349,0.0000
C02310=1970.210,342.503,-503.612,89.0032,-0.1948,0.0057
C02311=1958.875,342.539,-503.612,89.6220,-0.4755,0.0057
C02312=1953.389,342.556,-503.612,90.4528,-1.2146,-0.0114
C02313=1927.791,342.573,-503.612,89.8684,0.3838,0.0000
C02314=1936.371,342.595,-503.612,90.0804,0.1718,0.0000
C02315=1927.557,342.619,-503.612,89.9371,0.8708,0.0000
C02316=1971.976,342.660,-503.612,90.1033,-0.3208,0.0000
C02317=1985.894,342.701,-503.612,90.3783,0.0802,0.0000
C02318=1933.723,342.718,-503.612,91.1346,0.8078,0.0171
C02319=1983.719,342.754,-503.612,87.9891,-1.4209,0.0515
C02320=1967.433,342.769,-503.612,88.9173,0.5786,-0.0114
C02321=1971.507,342.796,-503.612,88.5105,0.1260,-0.0057
C02322=1978.383,342.823,-503.612,89.5647,-0.0572,0.0000
C02323=1956.724,342.919,-503.612,89.7194,-0.1948,0.0000
C02324=1964.207,342.910,-553.612,89.4559,0.0229,0.0000
C02325=1956.730,342.867,-553.612,89.4157,0.7333,-0.0057
C02326=1949.078,342.842,-553.612,90.3325,0.3724,0.0000
C02327=1964.487,342.819,-553.612,90.0976,-1.0599,0.0000
C02328=1980.017,342.771,-553.612,90.2981,-0.7333,-0.0057
C02329=1979.608,342.747,-553.612,90.8080,-0.0916,0.0000
C02330=1991.957,342.725,-553.612,90.0002,0.0630,0.0000
C02331=1961.526,342.702,-553.612,89.8970,0.2692,0.0000
C02332=1983.865,342.684,-553.612,90.1549,-0.3838,0.0000
C02333=1962.726,342.669,-553.612,90.9570,-0.3437,-0.0057
C02334=1991.699,342.655,-553.612,89.1866,-0.2177,0.0057
C02335=1935.378,342.638,-553.612,90.7507,0.3724,0.0057
C02336=1989.062,342.618,-553.612,89.9371,-0.0114,0.0000
C02337=1998.951,342.595,-553.612,89.9314,-1.1401,0.0000
C02338=1957.989,342.568,-553.612,90.9169,0.3036,0.0057
C02339=1958.395,342.561,-553.612,91.4211,-0.0229,0.0000
C02340=1912.496,342.529,-553.612,90.4700,0.5099,0.0057
C02341=1994.182,342.510,-553.612,91.9138,-0.1948,-0.0057
C02342=1980.976,342.483,-553.612,91.2034,-0.3093,-0.0057
C02343=2004.766,342.464,-553.612,90.3038,-1.4323,-0.0057
C02344=2003.375,342.426,-553.612,90.5101,-0.6359,-0.0057
C02345=1952.385,342.402,-553.612,91.7821,0.7505,0.0229
C02346=1910.094,342.379,-553.612,90.3611,1.7933,0.0114
C02347=2015.315,342.351,-553.612,91.1919,-1.3006,-0.0286
C02348=1938.235,342.325,-553.612,91.3867,-0.2406,-0.0057
C02349=2013.285,342.308,-553.612,90.8481,-0.8078,-0.0114
C02350=2019.297,342.292,-553.612,89.6048,-0.6932,0.0057
C02351=2008.569,342.270,-553.612,91.3352,-0.6359,-0.0171
C02352=2018.916,342.222,-553.612,90.8023,-0.7620,-0.0114
C02353=1979.372,342.200,-553.612,91.0831,-0.8651,-0.0171
C02354=2016.598,342.168,-553.612,90.6992,-1.4553,-0.0171
C02355=2006.372,342.140,-553.612,91.9597,-0.8537,-0.0286
C02356=2030.472,342.119,-553.612,89.1579,-0.9281,0.0114
C02357=1890.291,342.068,-553.612,90.0002,0.7964,0.0000
C02358=1897.591,342.045,-553.612,91.2435,1.5928,0.0343
C02359=2045.790,342.020,-553.612,89.3012,-0.4182,0.0057
C02360=2045.991,341.966,-553.612,91.0831,-0.4698,-0.0114
C02361=2038.443,341.945,-553.612,90.1205,-0.4182,0.0000
C02362=2042.479,341.930,-553.612,91.8050,-0.0744,0.0000
C02363=1898.504,341.915,-553.612,89.9429,1.8277,0.0000
C02364=2032.882,341.883,-553.612,91.7649,-1.4266,-0.0458
C02365=2015.277,341.840,-553.612,91.2893,-1.1802,-0.0286
C02366=1898.244,341.801,-553.612,91.4326,1.0026,0.0229
C02367=1893.562,341.768,-553.612,90.7507,1.0026,0.0114
C02368=1880.777,341.723,-553.612,90.4814,1.1688,0.0114
C02369=2046.840,341.707,-553.612,90.1606,-0.8250,0.0000
C02370=2069.878,341.676,-553.612,90.9169,-0.8422,-0.0114
C02371=2040.561,341.657,-553.612,91.9024,-0.9854,-0.0343
C02372=2052.105,341.625,-553.612,90.8138,-0.6932,-0.0114
C02373=1875.965,341.578,-553.612,90.8138,0.4526,0.0057
C02374=2082.093,341.573,-553.612,91.5414,-1.1516,-0.0286
C02375=1799.023,341.543,-553.612,90.6877,1.4152,0.0171
C02376=1860.945,341.526,-553.612,89.8283,0.9511,0.0000
C02377=2089.483,341.518,-553.612,90.6934,-0.7906,-0.0114
C02378=1867.784,341.508,-553.612,90.6419,0.2463,0.0000
C02379=1803.221,341.494,-553.612,90.0746,-0.8021,0.0000
C02380=1796.053,341.486,-553.612,90.1892,7.1104,0.0229
C02381=1851.170,341.469,-553.612,89.8856,0.5672,0.0000
C02382=2071.772,341.439,-553.612,90.9054,-1.3521,-0.0229
C02383=2066.800,341.418,-553.612,91.0028,-1.0370,-0.0171
C02384=2185.746,341.402,-553.612,89.8168,0.2234,0.0000
C02385=1808.857,341.395,-553.612,89.3012,-0.5557,0.0057
C02386=1861.348,341.384,-553.612,89.9429,0.9511,0.0000
C02387=1794.346,341.374,-553.612,92.6358,14.2895,0.6531
C02388=2058.599,341.362,-553.612,90.4299,-0.7219,-0.0057
C02389=2172.169,341.353,-553.612,90.8252,0.4010,0.0057
C02390=2052.220,341.343,-553.612,90.5731,-0.8021,-0.0057
C02391=1831.522,341.336,-553.612,89.8856,-0.0343,0.0000
C02392=1806.243,341.327,-553.612,89.6908,-0.3953,0.0000
C02393=2094.196,341.319,-553.612,90.3611,-0.9281,-0.0057
C02394=1830.253,341.299,-553.612,89.8741,-0.0286,0.0000
C02395=2095.532,341.289,-553.612,91.1747,-1.4094,-0.0286
C02396=1836.079,341.278,-553.612,90.0116,0.0229,0.0000
C02397=2177.034,341.269,-553.612,90.3726,1.7647,0.0114
C02398=2070.756,341.248,-553.612,91.0659,-0.6703,-0.0114
C02399=2178.247,341.240,-553.612,90.1434,0.6589,0.0000
C02400=1860.429,341.235,-553.612,90.7450,4.3258,0.0572
C02401=2155.399,341.221,-553.612,91.0716,-0.1776,-0.0057
C02402=1850.372,341.199,-553.612,90.4757,0.4411,0.0057
C02403=1794.823,341.170,-553.612,90.7908,14.3182,0.1948
C02404=1827.853,341.157,-553.612,90.6132,-0.2922,-0.0057
C02405=2165.438,341.146,-553.612,90.3611,0.2692,0.0000
C02406=2170.953,341.132,-553.612,90.4299,0.0859,0.0000
C02407=2090.251,341.116,-553.612,90.1778,-0.5614,0.0000
C02408=2079.914,341.095,-553.612,90.8882,-0.5500,-0.0057
C02409=2163.450,341.067,-553.612,90.6304,0.7505,0.0057
C02410=2079.593,341.045,-553.612,90.1606,0.6187,0.0000
C02411=2103.730,341.030,-553.612,91.4383,-0.3838,-0.0114
C02412=2173.328,341.004,-553.612,90.3554,1.1745,0.0057
C02413=2096.643,340.968,-553.612,90.3382,-0.2463,0.0000
C02414=2115.653,340.926,-553.612,90.4643,-0.5729,-0.0057
C02415=2172.555,340.907,-553.612,90.8080,1.4667,0.0229
C02416=2166.320,340.877,-553.612,90.7278,0.5271,0.0057
C02417=2102.683,340.848,-553.612,90.8711,-0.9568,-0.0171
C02418=2159.266,340.812,-553.612,89.9486,0.3380,0.0000
C02419=2124.739,340.747,-553.612,90.8653,0.0515,0.0000
C02420=2147.251,340.711,-553.612,90.4814,-0.1317,0.0000
C02421=2124.127,340.644,-553.612,90.4012,-0.2635,0.0000
C02422=2155.011,340.515,-553.612,90.7106,0.9224,0.0114
C02423=2135.657,340.072,-603.612,90.6992,0.7391,0.0114
C02424=2156.343,340.090,-603.612,91.0544,0.6130,0.0114
C02425=2142.360,340.162,-603.612,91.0200,0.6531,0.0114
C02426=2153.966,340.206,-603.612,90.9570,0.3380,0.0057
C02427=2118.636,340.235,-603.612,90.8023,-0.2922,-0.0057
C02428=2076.694,340.275,-603.612,91.3008,-1.0198,-0.0229
C02429=2112.962,340.298,-603.612,90.6705,-0.7448,-0.0114
C02430=2144.168,340.327,-603.612,91.3466,-0.2234,-0.0057
C02431=2061.348,340.347,-603.612,91.1346,-0.3552,-0.0057
C02432=2073.181,340.360,-603.612,90.9226,-1.0026,-0.0171
C02433=2167.096,340.394,-603.612,90.6132,0.7677,0.0057
C02434=2135.276,340.414,-603.612,90.7335,0.0114,0.0000
C02435=2108.758,340.447,-603.612,91.3581,-0.7563,-0.0171
C02436=2167.455,340.459,-603.612,90.3096,1.0657,0.0057
C02437=2072.723,340.483,-603.612,90.1033,-0.5614,0.0000
C02438=2170.625,340.498,-603.612,90.4241,1.1631,0.0114
C02439=2120.756,340.519,-603.612,90.9971,-0.2349,-0.0057
C02440=2089.944,340.532,-603.612,91.1117,-0.5958,-0.0114
C02441=2055.163,340.569,-603.612,91.1232,-0.6073,-0.0114
C02442=2155.478,340.589,-603.612,90.2580,0.1661,0.0000
C02443=2081.867,340.611,-603.612,91.3409,-0.3093,-0.0057
C02444=2166.000,340.634,-603.612,90.4012,1.2032,0.0057
C02445=2093.938,340.652,-603.612,90.7622,-0.5099,-0.0057
C02446=2069.645,340.675,-603.612,91.6617,-1.2547,-0.0343
C02447=2178.852,340.705,-603.612,90.2351,2.7158,0.0114
C02448=1874.120,340.733,-603.612,91.1174,0.0802,0.0000
C02449=2167.772,340.746,-603.612,89.4845,4.1596,-0.0401
C02450=2071.179,340.784,-603.612,91.3237,-1.0771,-0.0229
C02451=2026.257,340.804,-603.612,91.5930,0.1776,0.0057
C02452=2039.382,340.810,-603.612,90.9856,-0.8193,-0.0114
C02453=1845.616,340.815,-603.612,90.2408,-0.3036,0.0000
C02454=2098.545,340.841,-603.612,90.3325,-0.3724,0.0000
C02455=1834.963,340.847,-603.612,90.7049,0.0057,0.0000
C02456=2182.533,340.865,-603.612,90.6018,2.3949,0.0229
C02457=1827.332,340.906,-603.612,90.3267,-0.9110,-0.0057
C02458=2009.358,340.930,-603.612,92.9681,0.7964,0.0401
C02459=1828.273,340.940,-603.612,90.6018,-0.5042,-0.0057
C02460=2189.959,340.945,-603.612,90.5788,-8.1130,-0.0802
C02461=1826.229,340.967,-603.612,90.0059,-0.6073,0.0000
C02462=2173.349,340.985,-603.612,90.2981,1.6902,0.0114
C02463=1862.164,340.998,-603.612,91.1690,0.7448,0.0171
C02464=1902.966,341.006,-603.612,91.4326,0.5271,0.0114
C02465=1896.874,341.026,-603.612,90.9112,0.6302,0.0114
C02466=1843.071,341.041,-603.612,90.5788,-0.0687,0.0000
C02467=1821.811,341.061,-603.612,90.2293,-0.3151,0.0000
C02468=2040.528,341.073,-603.612,91.9310,-0.8537,-0.0286
C02469=2030.809,341.086,-603.612,90.5617,-0.5557,-0.0057
C02470=1922.128,341.098,-603.612,91.6789,0.2349,0.0057
C02471=1913.531,341.101,-603.612,91.0659,0.4297,0.0057
C02472=1816.196,341.117,-603.612,89.8168,-1.6386,0.0057
C02473=1892.901,341.129,-603.612,91.2836,-0.1317,-0.0057
C02474=1855.602,341.155,-603.612,90.5674,0.7219,0.0057
C02475=1813.245,341.168,-603.612,89.3986,-1.1287,0.0114
C02476=2041.678,341.179,-603.612,90.2236,-1.0141,-0.0057
C02477=2186.206,341.193,-603.612,90.2752,-1.5928,-0.0057
C02478=1929.570,341.202,-603.612,91.9310,0.5844,0.0171
C02479=1833.615,341.217,-603.612,89.7022,0.7161,-0.0057
C02480=2020.591,341.222,-603.612,91.6503,-0.4812,-0.0114
C02481=1884.225,341.244,-603.612,90.7221,1.0886,0.0114
C02482=1898.398,341.257,-603.612,91.1633,0.8479,0.0171
C02483=2014.799,341.274,-603.612,91.5242,-0.1948,-0.0057
C02484=1908.938,341.295,-603.612,90.9284,0.6016,0.0114
C02485=2004.014,341.322,-603.612,91.0544,-0.9568,-0.0171
C02486=2007.317,341.344,-603.612,91.9368,-1.0828,-0.0343
C02487=1886.600,341.355,-603.612,91.0831,1.1172,0.0229
C02488=1870.568,341.370,-603.612,90.9742,0.5042,0.0057
C02489=1934.460,341.379,-603.612,91.2435,0.5958,0.0114
C02490=1959.958,341.384,-603.612,91.3237,-0.2578,-0.0057
C02491=1799.058,341.402,-603.612,90.0173,2.3032,0.0000
C02492=2016.771,341.442,-603.612,91.1232,-0.2463,-0.0057
C02493=1973.170,341.456,-603.612,92.0456,-0.6417,-0.0229
C02494=1987.390,341.477,-603.612,90.9054,-0.3953,-0.0057
C02495=1944.689,341.484,-603.612,91.6847,-0.1432,-0.0057
C02496=1886.880,341.528,-603.612,91.1575,1.0370,0.0229
C02497=1896.840,341.582,-603.612,91.0315,0.6130,0.0114
C02498=2036.002,341.600,-603.612,90.2981,-1.0026,-0.0057
C02499=1926.992,341.647,-603.612,91.5357,0.7505,0.0229
C02500=1904.287,341.672,-603.612,91.1633,0.7734,0.0171
C02501=1922.547,341.690,-603.612,91.3180,0.5443,0.0114
C02502=2010.209,341.710,-603.612,91.0429,-0.8136,-0.0171
C02503=1993.488,341.734,-603.612,90.9570,-0.1718,0.0000
C02504=1988.105,341.792,-603.612,90.8023,0.0916,0.0000
C02505=2019.868,341.819,-603.612,90.6018,-0.4239,-0.0057
C02506=1974.252,341.856,-603.612,91.8795,-0.6187,-0.0229
C02507=1935.427,341.914,-603.612,91.2034,0.2578,0.0057
C02508=1994.529,341.953,-603.612,91.3409,-0.1489,-0.0057
C02509=1978.104,342.052,-603.612,92.3550,-0.8422,-0.0343
C02510=2001.864,342.090,-603.612,90.7049,-1.2490,-0.0171
C02511=1961.792,342.129,-603.612,90.9054,-0.2807,-0.0057
C02512=1968.211,342.175,-603.612,91.1747,0.0515,0.0000
C02513=1995.375,342.226,-603.612,90.3153,-0.2692,0.0000
C02514=1959.702,342.364,-603.612,91.3753,-0.2750,-0.0057
C02515=1799.585,341.481,-653.612,89.8627,1.5240,-0.0057
C02516=1797.490,341.408,-653.612,89.5876,4.7039,-0.0343
C02517=1798.072,341.332,-653.612,89.5475,4.3773,-0.0343
C02518=1813.001,341.180,-653.612,90.3096,-1.0886,-0.0057
C02519=1809.005,341.137,-653.612,90.3554,-1.7990,-0.0114
C02520=1795.303,341.117,-653.612,90.8309,12.9316,0.1833
C02521=1818.726,341.080,-653.612,89.4215,-1.4667,0.0171
C02522=1939.900,341.014,-653.612,91.6789,0.1833,0.0057
C02523=1794.649,340.970,-653.612,91.1919,19.4118,0.3953
C02524=1920.963,340.929,-653.612,90.4299,0.2750,0.0000
C02525=1993.976,340.898,-653.612,91.6159,-0.6932,-0.0171
C02526=1907.219,340.884,-653.612,91.4555,0.4297,0.0114
C02527=1822.301,340.862,-653.612,90.4356,-1.1917,-0.0114
C02528=1952.703,340.836,-653.612,91.8852,0.4182,0.0114
C02529=1900.084,340.808,-653.612,90.2924,0.5213,0.0000
C02530=2005.588,340.801,-653.612,91.1690,-0.2979,-0.0057
C02531=1920.569,340.791,-653.612,91.8050,0.2291,0.0057
C02532=1993.982,340.779,-653.612,94.1083,0.6818,0.0515
C02533=1964.959,340.769,-653.612,93.8676,0.0343,0.0000
C02534=1960.912,340.748,-653.612,90.4299,-0.1833,0.0000
C02535=1944.714,340.712,-653.612,90.5788,-0.2349,0.0000
C02536=1861.279,340.701,-653.612,91.7362,-0.5385,-0.0171
C02537=1877.044,340.694,-653.612,90.5960,-0.7047,-0.0057
C02538=1851.847,340.683,-653.612,90.2752,0.5729,0.0000
C02539=1848.928,340.657,-653.612,90.2866,-0.3437,0.0000
C02540=2186.041,340.631,-653.612,90.2408,1.2948,0.0057
C02541=1837.769,340.620,-653.612,90.2122,-0.8938,-0.0057
C02542=2179.220,340.605,-653.612,89.9887,2.3949,0.0000
C02543=2181.886,340.594,-653.612,90.4986,2.8647,0.0229
C02544=1884.869,340.587,-653.612,91.1232,0.3666,0.0057
C02545=1929.227,340.579,-653.612,91.7305,0.0286,0.0000
C02546=1935.934,340.554,-653.612,91.3810,0.4239,0.0114
C02547=1975.026,340.541,-653.612,91.0601,0.0916,0.0000
C02548=1983.594,340.531,-653.612,91.4899,-0.3036,-0.0057
C02549=1957.244,340.515,-653.612,92.3321,-0.2463,-0.0114
C02550=2181.325,340.501,-653.612,89.4329,2.6470,-0.0286
C02551=2029.531,340.495,-653.612,91.3581,-0.5672,-0.0114
C02552=2008.733,340.470,-653.612,90.1778,-0.8880,0.0000
C02553=1931.404,340.449,-653.612,90.9742,0.1317,0.0000
C02554=1879.484,340.436,-653.612,90.4528,-0.0916,0.0000
C02555=2187.220,340.422,-653.612,92.4581,-2.0855,-0.0916
C02556=1907.734,340.397,-653.612,90.4700,0.3896,0.0057
C02557=2042.416,340.383,-653.612,91.4612,0.5786,0.0171
C02558=1896.512,340.364,-653.612,90.5044,0.1317,0.0000
C02559=1863.838,340.358,-653.612,90.4643,-0.2234,0.0000
C02560=2027.516,340.350,-653.612,90.9226,-0.8078,-0.0114
C02561=2190.389,340.335,-653.612,92.2805,-12.6509,-0.4984
C02562=1857.257,340.319,-653.612,90.5445,-0.6359,-0.0057
C02563=1871.454,340.309,-653.612,90.3038,-0.3437,0.0000
C02564=2172.656,340.290,-653.612,89.9486,1.3865,0.0000
C02565=2168.784,340.287,-653.612,90.8768,1.0886,0.0171
C02566=1916.606,340.274,-653.612,91.0888,0.1088,0.0000
C02567=1899.370,340.264,-653.612,90.3096,-0.4297,0.0000
C02568=2021.925,340.239,-653.612,91.2836,-0.3666,-0.0057
C02569=1962.435,340.223,-653.612,90.9799,0.1260,0.0000
C02570=1932.220,340.197,-653.612,90.9226,0.0057,0.0000
C02571=2017.464,340.184,-653.612,91.0258,0.0515,0.0000
C02572=2167.720,340.167,-653.612,91.1232,0.6417,0.0114
C02573=1877.825,340.144,-653.612,89.7767,-0.5385,0.0000
C02574=2038.197,340.130,-653.612,90.6705,-0.2578,-0.0057
C02575=2080.355,340.103,-653.612,90.4471,-0.1145,0.0000
C02576=1931.894,340.092,-653.612,90.9455,0.4698,0.0057
C02577=2072.300,340.076,-653.612,91.3867,-0.2177,-0.0057
C02578=2165.460,340.065,-653.612,90.3840,0.7792,0.0057
C02579=2065.765,340.053,-653.612,90.6075,-0.0572,0.0000
C02580=2148.257,340.032,-653.612,90.7966,-0.2807,-0.0057
C02581=2048.677,340.015,-653.612,90.1606,-0.3609,0.0000
C02582=2152.310,339.998,-653.612,88.3558,0.0114,0.0000
C02583=2149.685,339.989,-653.612,90.6247,0.5729,0.0057
C02584=1970.078,339.973,-653.612,90.0288,0.4354,0.0000
C02585=2062.637,339.953,-653.612,90.6361,0.2234,0.0000
C02586=2096.443,339.933,-653.612,91.4268,0.0286,0.0000
C02587=2073.972,339.918,-653.612,89.9371,-0.2979,0.0000
C02588=2130.009,339.895,-653.612,90.5101,0.3781,0.0057
C02589=2162.184,339.887,-653.612,90.0403,0.9281,0.0000
C02590=2087.105,339.866,-653.612,90.6361,-0.3036,-0.0057
C02591=2156.929,339.855,-653.612,89.6392,0.5271,-0.0057
C02592=2072.996,339.844,-653.612,90.9169,0.1088,0.0000
C02593=2141.594,339.830,-653.612,91.1117,1.5985,0.0286
C02594=2161.208,339.821,-653.612,90.4929,1.0084,0.0114
C02595=2028.181,339.808,-653.612,90.2465,-0.7448,-0.0057
C02596=2093.127,339.781,-653.612,90.8596,-0.3495,-0.0057
C02597=2124.221,339.766,-653.612,90.8882,0.0401,0.0000
C02598=2153.667,339.747,-653.612,90.5903,0.6187,0.0057
C02599=2093.380,339.739,-653.612,90.6018,-0.6130,-0.0057
C02600=2124.244,339.722,-653.612,90.3096,0.2177,0.0000
C02601=2083.703,339.682,-653.612,89.7366,-0.0401,0.0000
C02602=2127.061,339.664,-653.612,89.8856,0.3724,0.0000
C02603=2134.955,339.649,-653.612,88.2813,0.9511,-0.0286
C02604=2101.613,339.635,-653.612,90.2637,0.3380,0.0000
C02605=2118.165,339.608,-653.612,90.5445,0.0916,0.0000
C02606=2116.317,339.587,-653.612,90.9570,0.1661,0.0000
C02607=2128.394,339.554,-653.612,90.9341,-0.0974,0.0000
C02608=2114.039,339.509,-653.612,90.6533,0.0057,0.0000
C02609=2073.190,338.995,-703.612,90.5158,-0.1088,0.0000
C02610=2063.755,339.117,-703.612,90.7679,0.6130,0.0057
C02611=2093.591,339.162,-703.612,90.3439,0.5042,0.0057
C02612=2077.013,339.188,-703.612,89.2152,0.8651,-0.0114
C02613=2089.260,339.222,-703.612,90.8882,0.8479,0.0114
C02614=1995.708,339.241,-703.612,90.6304,-0.1317,0.0000
C02615=2081.808,339.252,-703.612,89.3241,0.9625,-0.0114
C02616=2023.063,339.266,-703.612,90.5330,-0.0630,0.0000
C02617=2029.208,339.277,-703.612,89.7767,0.1145,0.0000
C02618=1977.825,339.286,-703.612,90.4356,-0.3552,0.0000
C02619=2107.308,339.308,-703.612,90.5903,-0.2807,-0.0057
C02620=2117.358,339.319,-703.612,90.5617,0.1260,0.0000
C02621=2013.371,339.330,-703.612,89.8054,-0.1203,0.0000
C02622=2059.863,339.337,-703.612,90.4929,-0.0630,0.0000
C02623=2048.126,339.350,-703.612,90.9169,-0.0572,0.0000
C02624=2083.336,339.354,-703.612,90.9513,-0.1718,-0.0057
C02625=2037.648,339.368,-703.612,90.3325,0.0343,0.0000
C02626=2099.786,339.381,-703.612,89.8397,0.3953,0.0000
C02627=2040.439,339.396,-703.612,91.0315,-0.0343,0.0000
C02628=1982.033,339.410,-703.612,89.4845,-0.0916,0.0000
C02629=2066.113,339.417,-703.612,90.5731,-0.5672,-0.0057
C02630=2130.776,339.427,-703.612,89.8741,0.8995,0.0000
C02631=2125.115,339.438,-703.612,90.6132,-0.0515,0.0000
C02632=2075.552,339.453,-703.612,90.4814,-0.1145,0.0000
C02633=2042.672,339.464,-703.612,90.7278,0.4182,0.0057
C02634=2069.289,339.474,-703.612,89.8569,0.1661,0.0000
C02635=2058.758,339.483,-703.612,90.3325,0.0572,0.0000
C02636=2057.580,339.492,-703.612,90.0116,-1.0714,0.0000
C02637=2134.466,339.499,-703.612,89.6908,-0.1718,0.0000
C02638=2007.649,339.513,-703.612,90.4070,-0.0343,0.0000
C02639=2121.289,339.520,-703.612,90.6648,0.0229,0.0000
C02640=2139.914,339.533,-703.612,90.0288,0.6130,0.0000
C02641=2048.001,339.547,-703.612,90.5330,-0.5099,-0.0057
C02642=2190.966,339.567,-703.612,90.1148,-14.5875,-0.0286
C02643=2134.176,339.577,-703.612,90.2866,0.0286,0.0000
C02644=2149.575,339.602,-703.612,89.8512,0.6073,0.0000
C02645=2146.144,339.608,-703.612,90.4585,0.4010,0.0057
C02646=2154.030,339.619,-703.612,90.6247,-0.5156,-0.0057
C02647=2156.547,339.633,-703.612,90.2637,0.7563,0.0057
C02648=1911.745,339.643,-703.612,89.5876,-0.7104,0.0057
C02649=1997.455,339.656,-703.612,91.1461,-0.5099,-0.0114
C02650=1962.991,339.666,-703.612,90.6763,-0.4010,-0.0057
C02651=2020.153,339.671,-703.612,92.4811,0.0286,0.0000
C02652=2151.746,339.683,-703.612,90.2809,0.3896,0.0000
C02653=1978.709,339.695,-703.612,91.5300,-0.4812,-0.0114
C02654=2191.127,339.708,-703.612,91.1232,-14.0546,-0.2750
C02655=2163.110,339.716,-703.612,90.5044,0.3896,0.0057
C02656=1903.782,339.744,-703.612,90.1377,-0.6474,0.0000
C02657=1940.902,339.759,-703.612,90.5617,-0.0229,0.0000
C02658=2183.988,339.776,-703.612,90.4929,-0.3380,-0.0057
C02659=1960.082,339.794,-703.612,90.8252,-0.1718,0.0000
C02660=1883.595,339.814,-703.612,89.8397,-0.8136,0.0000
C02661=1912.900,339.833,-703.612,90.7565,-0.0744,0.0000
C02662=2178.615,339.846,-703.612,90.0746,1.3407,0.0000
C02663=2024.628,339.859,-703.612,90.9455,-0.2578,-0.0057
C02664=2178.476,339.872,-703.612,92.3206,-0.3093,-0.0114
C02665=2183.640,339.884,-703.612,91.5300,2.6871,0.0744
C02666=2174.707,339.907,-703.612,91.3523,1.3006,0.0286
C02667=1897.922,339.912,-703.612,89.3355,0.5042,-0.0057
C02668=1933.132,339.928,-703.612,90.9742,-0.0229,0.0000
C02669=1878.689,339.963,-703.612,90.2122,-1.1573,-0.0057
C02670=1895.861,339.983,-703.612,90.6648,-0.1031,0.0000
C02671=1902.499,340.024,-703.612,91.7591,0.3724,0.0114
C02672=1936.508,340.046,-703.612,90.7335,0.8078,0.0114
C02673=1947.976,340.058,-703.612,90.8882,-0.1375,0.0000
C02674=1883.597,340.066,-703.612,90.2924,-0.8880,-0.0057
C02675=2183.839,340.085,-703.612,90.8424,2.1371,0.0286
C02676=1917.888,340.119,-703.612,90.2924,0.1661,0.0000
C02677=1873.671,340.134,-703.612,90.0689,-0.4812,0.0000
C02678=2183.708,340.173,-703.612,90.0746,0.8537,0.0000
C02679=1859.955,340.209,-703.612,90.4413,-1.5183,-0.0114
C02680=1876.642,340.250,-703.612,90.7335,-0.4927,-0.0057
C02681=2185.258,340.280,-703.612,91.0945,0.0687,0.0000
C02682=1857.611,340.327,-703.612,89.6277,-0.5271,0.0057
C02683=1852.308,340.478,-703.612,89.7423,-1.2834,0.0057
C02684=1844.337,340.522,-703.612,90.0689,-0.8136,0.0000
C02685=1839.074,340.629,-703.612,90.1606,-1.1631,-0.0057
C02686=1828.744,340.737,-703.612,89.7251,-0.3151,0.0000
C02687=1825.416,340.774,-703.612,90.2924,-0.7505,-0.0057
C02688=1794.825,340.931,-703.612,89.6220,19.3086,-0.1260
C02689=1816.931,341.031,-703.612,89.6564,-1.2146,0.0057
C02690=1818.991,341.110,-703.612,89.7710,-1.9767,0.0057
C02691=1795.182,341.178,-703.612,85.9551,15.9855,-1.1172
C02692=1805.178,341.310,-703.612,89.5590,-1.5355,0.0114
C02693=1809.277,341.405,-703.612,89.2439,-1.4495,0.0171
C02694=1798.100,341.483,-703.612,88.8485,4.3487,-0.0859
C02695=1799.488,341.555,-703.612,90.3840,0.1317,0.0000
C02696=1799.967,341.624,-753.612,90.3955,1.1688,0.0057
C02697=1803.673,341.530,-753.612,91.1117,-1.6042,-0.0286
C02698=1804.957,341.437,-753.612,88.6709,-0.9797,0.0229
C02699=1807.130,341.404,-753.612,89.6678,-1.0771,0.0057
C02700=1813.473,341.329,-753.612,89.7309,-1.1745,0.0057
C02701=1810.931,341.258,-753.612,90.0059,-1.7016,0.0000
C02702=1820.076,341.165,-753.612,90.2637,-0.4640,0.0000
C02703=1829.211,341.091,-753.612,90.3267,-0.9797,-0.0057
C02704=1827.450,340.976,-753.612,89.7481,-1.2719,0.0057
C02705=1827.531,340.915,-753.612,90.5158,-0.7849,-0.0057
C02706=1841.303,340.791,-753.612,89.5475,-1.1860,0.0114
C02707=1844.090,340.649,-753.612,89.6793,-1.3063,0.0057
C02708=1848.833,340.492,-753.612,89.8856,-1.4094,0.0000
C02709=1855.718,340.392,-753.612,89.4272,-1.0714,0.0114
C02710=1859.766,340.307,-753.612,89.9887,-1.5011,0.0000
C02711=1862.410,340.204,-753.612,89.9601,-1.8162,0.0000
C02712=1863.830,340.143,-753.612,89.4788,-1.3579,0.0114
C02713=1881.470,340.082,-753.612,89.9715,-0.4297,0.0000
C02714=1887.120,340.005,-753.612,89.5303,-0.4010,0.0057
C02715=1889.231,339.927,-753.612,89.9142,-0.3036,0.0000
C02716=1888.561,339.891,-753.612,90.1205,-1.3349,0.0000
C02717=1902.175,339.843,-753.612,90.0575,-0.3208,0.0000
C02718=1899.627,339.779,-753.612,90.2924,-0.8651,-0.0057
C02719=1897.177,339.749,-753.612,89.6850,-0.4984,0.0000
C02720=2160.074,339.715,-753.612,90.3669,0.0572,0.0000
C02721=1899.047,339.686,-753.612,89.5819,-0.4068,0.0057
C02722=2191.473,339.658,-753.612,89.8569,-17.9278,0.0458
C02723=1908.888,339.625,-753.612,90.2580,-0.6589,-0.0057
C02724=2178.824,339.612,-753.612,89.7423,1.2261,-0.0057
C02725=1918.495,339.594,-753.612,89.6965,-0.5156,0.0000
C02726=2163.106,339.570,-753.612,90.5330,0.1604,0.0000
C02727=2163.901,339.560,-753.612,90.0345,-0.5271,0.0000
C02728=1918.974,339.531,-753.612,90.2924,-0.2692,0.0000
C02729=2179.564,339.514,-753.612,90.4127,1.0084,0.0057
C02730=2153.582,339.502,-753.612,90.7851,0.1604,0.0000
C02731=1927.798,339.497,-753.612,89.7080,-0.7219,0.0057
C02732=1963.372,339.484,-753.612,90.4299,-0.8136,-0.0057
C02733=2153.419,339.472,-753.612,90.3439,0.3437,0.0000
C02734=1924.024,339.462,-753.612,90.1090,-0.6703,0.0000
C02735=2168.128,339.440,-753.612,89.8111,-0.2635,0.0000
C02736=2127.752,339.424,-753.612,89.6449,0.4068,0.0000
C02737=2157.929,339.408,-753.612,90.1319,0.4583,0.0000
C02738=2182.084,339.396,-753.612,89.4157,1.1401,-0.0114
C02739=1943.022,339.384,-753.612,90.5903,-0.6760,-0.0057
C02740=1943.388,339.372,-753.612,89.8913,-0.8250,0.0000
C02741=2146.933,339.357,-753.612,90.2122,0.2234,0.0000
C02742=1944.277,339.339,-753.612,89.7309,-0.1948,0.0000
C02743=2145.381,339.321,-753.612,90.5617,0.2635,0.0000
C02744=1955.529,339.311,-753.612,90.4299,-0.0974,0.0000
C02745=2126.821,339.291,-753.612,90.6075,0.1833,0.0000
C02746=1946.430,339.286,-753.612,89.7022,-0.2349,0.0000
C02747=1963.293,339.277,-753.612,88.9688,-0.4239,0.0057
C02748=1985.309,339.259,-753.612,91.2263,-0.4526,-0.0114
C02749=1961.859,339.246,-753.612,91.1919,-0.5672,-0.0114
C02750=2133.264,339.234,-753.612,89.7882,0.8823,-0.0057
C02751=2001.200,339.224,-753.612,90.0345,0.1661,0.0000
C02752=1953.498,339.214,-753.612,90.0059,0.2291,0.0000
C02753=2110.513,339.208,-753.612,89.6793,0.4927,0.0000
C02754=2010.070,339.200,-753.612,90.5387,-0.6073,-0.0057
C02755=2133.135,339.191,-753.612,90.8940,0.5385,0.0057
C02756=2014.725,339.180,-753.612,90.3611,0.0401,0.0000
C02757=2125.637,339.165,-753.612,90.2981,-0.1145,0.0000
C02758=2104.683,339.146,-753.612,90.3439,0.3036,0.0000
C02759=2129.776,339.141,-753.612,90.1549,0.8078,0.0000
C02760=2071.817,339.136,-753.612,91.1346,0.2807,0.0057
C02761=2057.477,339.112,-753.612,89.6105,1.3750,-0.0114
C02762=2061.228,339.100,-753.612,90.2695,-0.0687,0.0000
C02763=1975.866,339.086,-753.612,90.9054,-0.1661,0.0000
C02764=2041.824,339.079,-753.612,90.7966,-0.0401,0.0000
C02765=2058.845,339.075,-753.612,90.4070,0.8136,0.0057
C02766=2015.305,339.069,-753.612,89.7366,-1.0886,0.0057
C02767=1968.919,339.056,-753.612,91.2549,-0.5042,-0.0114
C02768=2054.725,339.041,-753.612,90.3554,0.2979,0.0000
C02769=2104.969,339.035,-753.612,90.0345,0.9167,0.0000
C02770=2082.812,339.026,-753.612,88.9746,0.3724,-0.0057
C02771=2027.650,339.018,-753.612,90.7565,-0.1833,0.0000
C02772=1998.073,339.007,-753.612,89.8970,-0.3437,0.0000
C02773=2074.825,338.992,-753.612,89.3584,1.1860,-0.0114
C02774=2089.149,338.987,-753.612,90.0517,-0.5901,0.0000
C02775=2053.323,338.978,-753.612,90.3325,-0.3323,0.0000
C02776=2097.125,338.974,-753.612,90.7049,-0.5786,-0.0057
C02777=2022.267,338.959,-753.612,90.3153,-0.2692,0.0000
C02778=2024.850,338.932,-753.612,91.3180,0.3552,0.0057
C02779=2085.333,338.914,-753.612,89.8913,0.1661,0.0000
C02780=2038.206,338.906,-753.612,89.9715,-0.3208,0.0000
C02781=2066.504,338.886,-753.612,90.1205,-0.0057,0.0000
C02782=2093.534,338.865,-753.612,89.8225,0.0916,0.0000
C02783=2058.436,338.801,-753.612,90.1319,-0.6760,0.0000
C02784=2073.063,338.735,-803.612,90.3439,-0.8078,-0.0057
C02785=2062.264,338.781,-803.612,89.3642,0.4812,-0.0057
C02786=2061.218,338.791,-803.612,89.5475,-0.2119,0.0000
C02787=1999.241,338.815,-803.612,88.7798,1.2605,-0.0286
C02788=2061.161,338.858,-803.612,89.2037,0.2750,-0.0057
C02789=2096.996,338.867,-803.612,88.8084,0.3724,-0.0057
C02790=2032.901,338.882,-803.612,89.9429,-0.3093,0.0000
C02791=2104.217,338.888,-803.612,91.1747,1.5985,0.0343
C02792=2019.781,338.898,-803.612,89.5876,0.2750,0.0000
C02793=2032.219,338.910,-803.612,89.5647,-0.0171,0.0000
C02794=2088.973,338.917,-803.612,90.1950,0.0515,0.0000
C02795=2038.272,338.924,-803.612,89.8340,-0.1776,0.0000
C02796=2014.609,338.933,-803.612,89.8627,-0.2521,0.0000
C02797=2100.091,338.939,-803.612,90.9742,-0.3151,-0.0057
C02798=2046.154,338.945,-803.612,90.8424,-0.8078,-0.0114
C02799=2077.330,338.949,-803.612,89.8569,-0.2864,0.0000
C02800=2071.967,338.953,-803.612,89.7423,0.1604,0.0000
C02801=1988.870,338.964,-803.612,90.1148,-0.5042,0.0000
C02802=2111.765,338.974,-803.612,89.9830,0.6016,0.0000
C02803=2118.654,338.987,-803.612,89.8283,0.0687,0.0000
C02804=2105.787,338.990,-803.612,90.4070,0.3093,0.0000
C02805=2049.676,338.996,-803.612,90.2351,-0.4870,0.0000
C02806=2122.801,339.002,-803.612,90.1434,0.5213,0.0000
C02807=1998.518,339.016,-803.612,89.9772,-0.1375,0.0000
C02808=2159.190,339.028,-803.612,90.3497,0.4469,0.0000
C02809=2102.381,339.034,-803.612,90.3669,0.4526,0.0057
C02810=2042.336,339.040,-803.612,89.8741,0.4297,0.0000
C02811=2113.548,339.047,-803.612,90.1434,0.0515,0.0000
C02812=2131.010,339.059,-803.612,89.4845,0.4526,-0.0057
C02813=1990.465,339.066,-803.612,90.6705,-0.5213,-0.0057
C02814=2154.185,339.079,-803.612,90.4929,0.2578,0.0000
C02815=2103.755,339.090,-803.612,89.8798,0.3495,0.0000
C02816=1978.876,339.102,-803.612,89.6048,-0.1604,0.0000
C02817=2108.690,339.109,-803.612,89.7366,0.5213,0.0000
C02818=2117.282,339.118,-803.612,89.1579,0.9854,-0.0171
C02819=2167.864,339.126,-803.612,90.4700,0.4698,0.0057
C02820=1968.699,339.144,-803.612,89.9371,-0.5213,0.0000
C02821=1980.830,339.149,-803.612,89.5533,-0.6359,0.0057
C02822=2012.761,339.158,-803.612,89.3126,-0.2349,0.0000
C02823=1979.519,339.173,-803.612,89.2152,-0.3953,0.0057
C02824=2133.101,339.181,-803.612,90.0689,-0.4870,0.0000
C02825=2139.307,339.203,-803.612,90.2007,0.7219,0.0000
C02826=2189.894,339.212,-803.612,90.8653,-6.1077,-0.0916
C02827=2164.407,339.218,-803.612,90.7794,-0.1317,0.0000
C02828=1973.765,339.226,-803.612,88.9975,0.0515,0.0000
C02829=1963.063,339.232,-803.612,89.7939,-0.1203,0.0000
C02830=2140.823,339.248,-803.612,89.2840,0.6932,-0.0114
C02831=1966.561,339.257,-803.612,90.4413,-0.7219,-0.0057
C02832=2146.546,339.275,-803.612,89.7366,0.4698,0.0000
C02833=1944.493,339.305,-803.612,89.6507,-0.3953,0.0000
C02834=2164.597,339.332,-803.612,90.9341,0.6818,0.0114
C02835=2179.742,339.345,-803.612,90.6304,1.9537,0.0229
C02836=1959.256,339.353,-803.612,89.8455,-0.3151,0.0000
C02837=1951.206,339.375,-803.612,90.2523,-0.6359,0.0000
C02838=1940.398,339.403,-803.612,89.8397,-0.5901,0.0000
C02839=1952.858,339.430,-803.612,90.2695,-0.1031,0.0000
C02840=1940.391,339.450,-803.612,90.1720,-0.6760,0.0000
C02841=1925.004,339.506,-803.612,90.0002,-0.4411,0.0000
C02842=1931.783,339.527,-803.612,89.8397,-0.2578,0.0000
C02843=1915.754,339.565,-803.612,89.9142,-0.2922,0.0000
C02844=1925.891,339.622,-803.612,89.5418,-0.5385,0.0057
C02845=1939.013,339.694,-803.612,89.8970,-0.0343,0.0000
C02846=1916.706,339.756,-803.612,90.0173,-0.8479,0.0000
C02847=1906.137,339.800,-803.612,89.6850,-0.7620,0.0057
C02848=1908.335,339.879,-803.612,89.4559,-0.4984,0.0057
C02849=1891.927,339.960,-803.612,89.7481,-0.9854,0.0057
C02850=1898.280,340.042,-803.612,89.5533,-0.9854,0.0057
C02851=1878.249,340.138,-803.612,90.0173,-1.2547,0.0000
C02852=1890.381,340.206,-803.612,90.6018,0.4068,0.0057
C02853=1874.073,340.238,-803.612,89.7595,-1.2032,0.0057
C02854=1872.070,340.338,-803.612,89.7423,-0.5271,0.0000
C02855=1878.439,340.425,-803.612,89.9830,-0.8422,0.0000
C02856=1863.563,340.545,-803.612,89.8111,-1.1573,0.0057
C02857=1858.204,340.602,-803.612,90.0517,-1.0370,0.0000
C02858=1846.137,340.776,-803.612,89.3756,-1.0485,0.0114
C02859=1846.450,340.848,-803.612,89.9772,-1.0084,0.0000
C02860=1839.612,340.979,-803.612,89.1465,-0.3552,0.0057
C02861=1829.812,341.022,-803.612,89.8684,-0.8594,0.0000
C02862=1794.925,341.065,-803.612,91.1002,14.6104,0.2807
C02863=1837.928,341.117,-803.612,89.4673,-0.6589,0.0057
C02864=1824.256,341.181,-803.612,89.5647,-0.6760,0.0057
C02865=1817.402,341.262,-803.612,89.4501,-1.3120,0.0114
C02866=1817.372,341.325,-803.612,90.1663,-1.1344,-0.0057
C02867=1808.346,341.423,-803.612,89.8225,-1.2719,0.0057
C02868=1812.505,341.463,-803.612,89.5762,-1.1802,0.0114
C02869=1798.014,341.534,-803.612,90.2179,5.4602,0.0229
C02870=1798.394,341.571,-803.612,90.4528,4.4977,0.0343
C02871=1798.782,341.649,-803.612,90.7335,3.2544,0.0401
C02872=1798.679,341.821,-853.612,89.0892,2.3663,-0.0401
C02873=1801.796,341.691,-853.612,90.3840,-0.3323,0.0000
C02874=1803.834,341.604,-853.612,91.3581,-1.9767,-0.0458
C02875=1797.252,341.515,-853.612,93.7187,6.8353,0.4411
C02876=1811.298,341.443,-853.612,90.4814,-1.9996,-0.0171
C02877=1813.044,341.369,-853.612,90.0746,-1.9308,0.0000
C02878=1814.433,341.317,-853.612,90.5101,-1.6730,-0.0171
C02879=1816.535,341.199,-853.612,90.0575,-0.8938,0.0000
C02880=1822.945,341.133,-853.612,89.6850,-1.2204,0.0057
C02881=1817.392,341.111,-853.612,90.4012,-1.0771,-0.0057
C02882=1843.858,340.985,-853.612,89.8397,-1.2375,0.0057
C02883=1842.018,340.879,-853.612,90.4127,-1.2490,-0.0114
C02884=1843.463,340.784,-853.612,90.0173,-0.4354,0.0000
C02885=1850.351,340.762,-853.612,89.9543,-0.8880,0.0000
C02886=1858.825,340.665,-853.612,89.8111,-1.1573,0.0057
C02887=1864.859,340.596,-853.612,89.1350,-0.0114,0.0000
C02888=1864.700,340.570,-853.612,90.2924,-0.7964,-0.0057
C02889=1884.815,340.449,-853.612,89.5934,-0.4354,0.0057
C02890=1866.700,340.415,-853.612,90.9455,-0.7333,-0.0114
C02891=1875.256,340.323,-853.612,90.2924,-0.4812,0.0000
C02892=1889.321,340.299,-853.612,89.5762,-0.7391,0.0057
C02893=1891.341,340.243,-853.612,89.9085,-1.0714,0.0000
C02894=1897.280,340.165,-853.612,90.8481,-0.6359,-0.0114
C02895=1904.713,340.119,-853.612,89.2152,-0.3781,0.0057
C02896=1934.186,340.090,-853.612,89.4043,-1.0943,0.0114
C02897=1904.887,340.006,-853.612,89.4444,-0.5729,0.0057
C02898=1913.416,339.981,-853.612,89.7538,-0.1031,0.0000
C02899=1924.127,339.912,-853.612,90.6075,-0.0458,0.0000
C02900=1952.628,339.828,-853.612,87.4047,-0.0630,0.0000
C02901=1953.652,339.784,-853.612,89.6507,-0.3896,0.0000
C02902=1947.297,339.762,-853.612,89.5876,0.0630,0.0000
C02903=1930.044,339.732,-853.612,89.3527,-0.5328,0.0057
C02904=1937.784,339.671,-853.612,88.8199,-1.0141,0.0229
C02905=1938.403,339.637,-853.612,89.9887,-0.4755,0.0000
C02906=2047.261,339.589,-853.612,77.3779,0.7677,-0.1718
C02907=1962.940,339.523,-853.612,90.0231,-1.0084,0.0000
C02908=1985.149,339.488,-853.612,88.3787,-0.4182,0.0114
C02909=1981.144,339.449,-853.612,90.0231,-0.6130,0.0000
C02910=1957.762,339.410,-853.612,89.6793,-0.3781,0.0000
C02911=1990.508,339.405,-853.612,90.1319,-0.1718,0.0000
C02912=2000.751,339.354,-853.612,89.3069,-0.2291,0.0000
C02913=1982.854,339.317,-853.612,88.7397,-0.4927,0.0114
C02914=2009.978,339.297,-853.612,89.5418,0.7677,-0.0057
C02915=2024.539,339.284,-853.612,90.0517,-0.2578,0.0000
C02916=2121.511,339.274,-853.612,88.4073,-0.3036,0.0057
C02917=2055.332,339.230,-853.612,90.1720,0.5328,0.0000
C02918=2038.502,339.213,-853.612,89.7538,-0.2521,0.0000
C02919=2083.289,339.197,-853.612,89.3527,0.0859,0.0000
C02920=1989.215,339.185,-853.612,89.0605,-0.3953,0.0057
C02921=2067.307,339.179,-853.612,89.9085,-0.8422,0.0000
C02922=2188.011,339.171,-853.612,90.6247,-5.0362,-0.0572
C02923=2006.290,339.150,-853.612,88.8542,0.3036,-0.0057
C02924=2087.059,339.135,-853.612,90.9398,-0.8422,-0.0114
C02925=2182.180,339.129,-853.612,89.7538,0.6531,0.0000
C02926=2165.223,339.123,-853.612,89.7366,0.7391,-0.0057
C02927=2179.411,339.116,-853.612,74.5704,-0.5385,0.1489
C02928=2178.774,339.105,-853.612,91.3294,-0.0229,0.0000
C02929=1995.124,339.097,-853.612,89.3584,-0.9682,0.0114
C02930=1998.114,339.089,-853.612,90.7966,-0.8537,-0.0114
C02931=2028.129,339.081,-853.612,91.6159,0.3323,0.0114
C02932=2071.745,339.075,-853.612,89.6105,-0.6073,0.0057
C02933=2107.939,339.069,-853.612,90.1606,0.1833,0.0000
C02934=2171.816,339.059,-853.612,89.6449,-0.4812,0.0057
C02935=2006.319,339.054,-853.612,90.7164,-0.4411,-0.0057
C02936=2061.621,339.046,-853.612,89.9371,-0.0974,0.0000
C02937=2092.362,339.039,-853.612,89.6507,-0.6875,0.0057
C02938=2127.230,339.028,-853.612,90.6533,-0.2979,-0.0057
C02939=2142.220,339.022,-853.612,90.0804,0.1317,0.0000
C02940=2050.404,339.012,-853.612,90.3669,-0.0974,0.0000
C02941=2017.120,339.008,-853.612,91.0086,-0.1489,0.0000
C02942=2097.055,339.005,-853.612,90.7450,-1.0828,-0.0114
C02943=2146.699,338.996,-853.612,90.1950,-0.3781,0.0000
C02944=2169.661,338.991,-853.612,90.2122,-0.5099,0.0000
C02945=2155.902,338.977,-853.612,90.3726,-0.2119,0.0000
C02946=2135.683,338.961,-853.612,89.8627,0.1432,0.0000
C02947=2045.946,338.948,-853.612,88.7798,0.8193,-0.0171
C02948=2091.307,338.939,-853.612,89.3928,-0.2521,0.0000
C02949=2072.474,338.934,-853.612,89.9944,-0.9568,0.0000
C02950=2109.023,338.915,-853.612,89.4960,-0.2234,0.0000
C02951=2059.240,338.906,-853.612,89.4215,-0.6760,0.0057
C02952=2189.032,338.897,-853.612,92.0915,-4.2513,-0.1546
C02953=2113.653,338.883,-853.612,90.8252,0.1890,0.0000
C02954=2114.931,338.865,-853.612,85.8061,-0.2349,0.0171
C02955=2141.954,338.841,-853.612,87.3244,-0.1375,0.0057
C02956=2158.166,338.775,-853.612,91.3638,-0.0687,0.0000
C02957=2182.832,338.676,-853.612,93.7702,-0.2692,-0.0171
C02958=2192.460,338.381,-853.612,92.8592,-14.6619,-0.7276
C02959=1845.943,-262.579,-444.761,-85.1357,-0.7964,179.9316
C02960=2103.620,-262.360,-444.761,-77.8477,0.3380,-179.9259
C02961=2106.924,-262.167,-444.761,-88.0865,0.2750,-179.9889
C02962=1869.037,-262.039,-444.761,-79.0223,1.2719,-179.7540
C02963=2042.284,-262.001,-444.761,-86.3218,1.4954,-179.9030
C02964=2099.976,-261.979,-444.761,-88.5792,1.3636,-179.9660
C02965=2077.569,-261.892,-444.761,-79.4749,-0.3781,179.9316
C02966=2056.224,-261.862,-444.761,-82.2480,-0.5557,179.9259
C02967=1929.876,-261.815,-444.761,-82.6548,1.3922,-179.8228
C02968=1953.938,-261.752,-444.761,-78.4035,-0.7849,179.8399
C02969=2043.564,-261.713,-444.761,-75.7221,-0.8021,179.7941
C02970=1974.190,-261.625,-444.761,-78.6671,-1.6730,179.6623
C02971=1921.842,-260.819,-494.761,-91.9654,0.1776,179.9946
C02972=1911.461,-260.905,-494.761,-92.2118,-0.5729,-179.9775
C02973=1866.999,-260.969,-494.761,-92.1659,-0.6130,-179.9775
C02974=1870.542,-261.046,-494.761,-91.8852,-0.3036,-179.9889
C02975=1916.503,-261.073,-494.761,-91.5357,0.4297,179.9889
C02976=1861.862,-261.137,-494.761,-92.0743,-0.9511,-179.9660
C02977=1937.964,-261.156,-494.761,-91.6961,0.1890,179.9946
C02978=1998.654,-261.175,-494.761,-91.1976,0.2062,179.9946
C02979=2020.094,-261.188,-494.761,-91.5357,-0.4239,-179.9889
C02980=1933.449,-261.219,-494.761,-92.8420,0.1546,179.9946
C02981=2024.472,-261.238,-494.761,-92.3436,-0.1203,-179.9946
C02982=2016.615,-261.241,-494.761,-91.5128,0.2635,179.9946
C02983=1957.998,-261.260,-494.761,-91.7420,0.4870,179.9832
C02984=2090.231,-261.293,-494.761,-91.8737,-0.1833,-179.9946
C02985=1857.870,-261.303,-494.761,-90.8997,0.2521,179.9946
C02986=1869.562,-261.332,-494.761,-91.1060,0.1604,179.9946
C02987=1956.272,-261.355,-494.761,-92.2691,-0.0630,-179.9946
C02988=1980.693,-261.373,-494.761,-91.2263,-0.5328,-179.9889
C02989=2081.434,-261.394,-494.761,-91.0601,-0.0229,-180.0004
C02990=1849.814,-261.409,-494.761,-91.6331,-0.1088,-179.9946
C02991=1898.632,-261.421,-494.761,-91.1518,-0.2005,-179.9946
C02992=2077.098,-261.431,-494.761,-91.1289,-0.6474,-179.9889
C02993=2080.090,-261.448,-494.761,-90.9971,-0.2692,-179.9946
C02994=1868.275,-261.460,-494.761,-91.6617,-0.6016,-179.9832
C02995=1897.656,-261.478,-494.761,-92.4983,2.1715,179.9030
C02996=2006.452,-261.495,-494.761,-91.9253,0.0057,180.0004
C02997=2097.180,-261.502,-494.761,-91.4326,0.2750,179.9946
C02998=2003.950,-261.515,-494.761,-90.3783,0.4182,179.9946
C02999=1974.234,-261.535,-494.761,-90.6591,-0.1432,-180.0004
C03000=2124.803,-261.548,-494.761,-91.6560,0.3036,179.9889
C03001=2094.531,-261.564,-494.761,-90.7679,0.5443,179.9946
C03002=2132.074,-261.573,-494.761,-91.2148,0.3380,179.9946
C03003=1884.756,-261.584,-494.761,-92.6472,-0.5672,-179.9717
C03004=1949.279,-261.598,-494.761,-90.6820,0.4984,179.9946
C03005=1986.413,-261.603,-494.761,-91.3294,0.9453,179.9775
C03006=2088.847,-261.615,-494.761,-90.6992,-0.6302,-179.9946
C03007=1907.677,-261.626,-494.761,-91.3237,-0.2177,-179.9946
C03008=2055.490,-261.635,-494.761,-90.4012,-0.0286,-180.0004
C03009=2026.414,-261.643,-494.761,-90.3611,-0.2692,-180.0004
C03010=2116.655,-261.651,-494.761,-90.5044,0.7505,179.9946
C03011=1933.336,-261.663,-494.761,-91.0487,0.1375,179.9946
C03012=2092.292,-261.669,-494.761,-92.2462,-0.0859,-179.9946
C03013=1945.953,-261.681,-494.761,-91.5930,0.3036,179.9889
C03014=2022.229,-261.689,-494.761,-90.5559,0.4927,179.9946
C03015=2193.443,-261.697,-494.761,-92.6300,-7.5630,-179.6566
C03016=1994.152,-261.709,-494.761,-90.9226,-0.7734,-179.9889
C03017=2117.856,-261.713,-494.761,-90.9455,0.8823,179.9832
C03018=2150.660,-261.719,-494.761,-91.1289,0.1260,180.0004
C03019=2026.671,-261.724,-494.761,-90.2122,0.6760,179.9946
C03020=2181.140,-261.730,-494.761,-89.4272,0.5786,-179.9946
C03021=1954.378,-261.737,-494.761,-90.8825,0.5844,179.9889
C03022=2027.263,-261.740,-494.761,-91.8737,-0.1546,-179.9946
C03023=1902.290,-261.748,-494.761,-91.2034,-0.0802,-180.0004
C03024=2083.758,-261.758,-494.761,-90.3325,-0.4984,-179.9946
C03025=1968.561,-261.766,-494.761,-89.2954,-0.4068,179.9946
C03026=2142.714,-261.772,-494.761,-90.8768,0.4526,179.9946
C03027=2013.614,-261.780,-494.761,-90.8367,-0.7964,-179.9889
C03028=2071.154,-261.790,-494.761,-91.1862,0.2750,179.9946
C03029=2077.380,-261.803,-494.761,-91.6445,0.5614,179.9832
C03030=1914.243,-261.809,-494.761,-90.4585,-0.6760,-179.9946
C03031=2162.444,-261.814,-494.761,-90.9169,0.2406,179.9946
C03032=1989.357,-261.816,-494.761,-90.6648,1.0771,179.9889
C03033=1909.275,-261.821,-494.761,-91.0143,0.0744,180.0004
C03034=2185.796,-261.830,-494.761,-89.9543,0.0515,-180.0004
C03035=1910.961,-261.834,-494.761,-91.4154,-0.1031,-179.9946
C03036=2170.544,-261.840,-494.761,-89.2381,-0.2005,179.9946
C03037=2169.153,-261.845,-494.761,-89.9715,-0.3151,180.0004
C03038=1865.804,-261.849,-494.761,-92.0972,0.6474,179.9775
C03039=1816.495,-261.851,-494.761,-91.8508,-0.8995,-179.9717
C03040=2024.305,-261.859,-494.761,-91.1117,0.2291,179.9946
C03041=2124.318,-261.865,-494.761,-90.9341,0.2463,179.9946
C03042=2080.300,-261.872,-494.761,-90.4643,-0.3552,-179.9946
C03043=2042.447,-261.881,-494.761,-90.2293,-0.3265,-180.0004
C03044=1805.058,-261.884,-494.761,-92.0972,-1.6042,-179.9431
C03045=2172.081,-261.890,-494.761,-90.5559,-0.0515,-180.0004
C03046=2035.399,-261.894,-494.761,-91.0716,0.2578,179.9946
C03047=2175.348,-261.898,-494.761,-90.8252,-0.3208,-179.9946
C03048=2190.438,-261.904,-494.761,-88.9860,-0.9511,179.9832
C03049=2165.547,-261.916,-494.761,-89.9830,-0.8537,180.0004
C03050=2188.317,-261.922,-494.761,-90.4528,0.3552,179.9946
C03051=1810.669,-261.930,-494.761,-91.7076,-1.3464,-179.9603
C03052=2095.544,-261.934,-494.761,-90.7622,-0.8708,-179.9889
C03053=2113.841,-261.939,-494.761,-88.8199,0.3151,-179.9946
C03054=2047.699,-261.949,-494.761,-90.3210,-0.1145,-180.0004
C03055=2038.089,-261.958,-494.761,-89.5131,-0.0057,180.0004
C03056=2022.620,-261.962,-494.761,-90.7049,-0.2922,-179.9946
C03057=2141.279,-261.973,-494.761,-90.1778,0.9511,179.9946
C03058=1879.830,-261.982,-494.761,-91.3466,0.3838,179.9889
C03059=2077.005,-262.004,-494.761,-90.3611,0.0286,180.0004
C03060=1821.697,-262.022,-494.761,-91.1805,-0.6875,-179.9832
C03061=2102.265,-262.033,-494.761,-90.0918,0.0916,180.0004
C03062=1839.440,-262.042,-494.761,-91.6388,0.1718,179.9946
C03063=1920.936,-262.050,-494.761,-84.4081,-0.9740,179.9030
C03064=1848.899,-262.065,-494.761,-89.3470,-1.7532,179.9775
C03065=1811.781,-262.089,-494.761,-91.1575,-1.0485,-179.9775
C03066=1805.613,-262.106,-494.761,-90.7679,-1.2834,-179.9832
C03067=2144.861,-262.140,-494.761,-89.7022,0.1661,-180.0004
C03068=1811.431,-262.204,-494.761,-90.1090,-1.2776,-179.9946
C03069=1863.241,-262.289,-494.761,-90.8825,-0.3036,-179.9946
C03070=1831.979,-262.356,-494.761,-93.2775,0.5042,179.9717
C03071=1796.446,-262.384,-494.761,-90.5788,5.8269,179.9431
C03072=1847.265,-262.436,-494.761,-91.0601,-1.1000,-179.9775
C03073=1818.793,-262.555,-494.761,-91.4899,-0.7964,-179.9775
C03074=1801.917,-262.590,-494.761,-91.8623,-1.3407,-179.9545
C03075=1806.287,-262.817,-494.761,-77.4180,-2.3262,179.4790
C03076=2193.404,-262.778,-544.761,-88.1667,1.7704,-179.9431
C03077=2189.447,-261.928,-544.761,-90.8138,4.3602,179.9373
C03078=2190.414,-261.848,-544.761,-90.6190,0.4182,179.9946
C03079=2184.051,-261.800,-544.761,-89.9601,-1.0485,180.0004
C03080=2181.482,-261.731,-544.761,-90.6934,0.6990,179.9889
C03081=2167.358,-261.706,-544.761,-90.6992,-0.1203,-180.0004
C03082=2171.713,-261.665,-544.761,-90.7622,0.1260,180.0004
C03083=2156.638,-261.640,-544.761,-91.0028,0.7448,179.9889
C03084=2139.836,-261.607,-544.761,-91.2893,0.1375,179.9946
C03085=1812.547,-261.579,-544.761,-91.2377,-1.7417,-179.9603
C03086=2171.946,-261.543,-544.761,-90.8596,1.2318,179.9832
C03087=2154.229,-261.503,-544.761,-91.0773,0.6990,179.9889
C03088=2173.622,-261.451,-544.761,-91.3180,0.6932,179.9832
C03089=1814.094,-261.418,-544.761,-90.7164,-1.0828,-179.9889
C03090=1805.093,-261.396,-544.761,-91.0659,-1.3980,-179.9717
C03091=2168.330,-261.378,-544.761,-90.9856,1.0255,179.9832
C03092=1836.531,-261.352,-544.761,-91.7133,-0.6245,-179.9832
C03093=2178.750,-261.297,-544.761,-90.4986,1.7417,179.9832
C03094=2100.472,-261.271,-544.761,-91.5128,0.2635,179.9946
C03095=2129.860,-261.209,-544.761,-92.2060,0.3552,179.9889
C03096=1809.421,-261.193,-544.761,-90.4929,-0.9339,-179.9946
C03097=2164.807,-261.175,-544.761,-90.3096,1.3063,179.9946
C03098=1821.197,-261.137,-544.761,-90.7393,-0.9167,-179.9889
C03099=2064.002,-261.115,-544.761,-91.4956,-0.0859,-180.0004
C03100=1837.038,-261.079,-544.761,-91.2893,-0.7964,-179.9832
C03101=2144.955,-261.059,-544.761,-91.5873,0.6703,179.9832
C03102=1816.312,-261.036,-544.761,-90.5731,-0.6818,-179.9946
C03103=2007.052,-261.008,-544.761,-91.2320,1.2891,179.9717
C03104=1815.077,-260.995,-544.761,-91.1060,-1.2547,-179.9775
C03105=2020.728,-260.981,-544.761,-91.6847,0.4010,179.9889
C03106=1935.614,-260.958,-544.761,-91.8279,0.3953,179.9889
C03107=1815.197,-260.941,-544.761,-89.5819,-1.9881,179.9832
C03108=2038.539,-260.917,-544.761,-92.3779,0.5844,179.9775
C03109=1995.584,-260.905,-544.761,-92.6931,0.3151,179.9832
C03110=1821.920,-260.891,-544.761,-91.1117,-1.1573,-179.9775
C03111=1972.452,-260.872,-544.761,-91.6617,0.1833,179.9946
C03112=1871.622,-260.855,-544.761,-91.8394,-0.2234,-179.9946
C03113=1992.617,-260.839,-544.761,-93.1629,0.0744,179.9946
C03114=2131.634,-260.824,-544.761,-91.6560,0.7792,179.9775
C03115=2035.438,-260.806,-544.761,-91.0372,-0.9339,-179.9832
C03116=2114.512,-260.763,-544.761,-91.4211,1.1287,179.9717
C03117=2078.864,-260.750,-544.761,-92.1717,0.2979,179.9889
C03118=2157.676,-260.733,-544.761,-91.3180,1.7074,179.9603
C03119=1866.480,-260.724,-544.761,-91.2263,-0.6474,-179.9889
C03120=1988.083,-260.707,-544.761,-91.8050,0.2463,179.9946
C03121=1978.238,-260.688,-544.761,-91.6732,0.7391,179.9775
C03122=1897.058,-260.662,-544.761,-92.8592,-1.3063,-179.9373
C03123=1825.113,-260.652,-544.761,-90.8768,-0.9511,-179.9832
C03124=2095.767,-260.644,-544.761,-91.6331,0.5443,179.9832
C03125=1876.881,-260.633,-544.761,-92.8363,0.7391,179.9660
C03126=2074.786,-260.610,-544.761,-92.1946,0.5614,179.9775
C03127=1924.829,-260.589,-544.761,-91.1862,-0.3896,-179.9946
C03128=2116.875,-260.582,-544.761,-91.9769,0.1432,179.9946
C03129=1842.483,-260.561,-544.761,-91.1633,-1.2433,-179.9775
C03130=2027.544,-260.536,-544.761,-91.8737,0.3437,179.9889
C03131=1850.823,-260.517,-544.761,-91.2435,-0.0687,-180.0004
C03132=1875.209,-260.495,-544.761,-91.9024,-0.1776,-179.9946
C03133=1971.870,-260.470,-544.761,-91.3638,0.3380,179.9946
C03134=1987.957,-260.444,-544.761,-91.1747,2.2345,179.9545
C03135=1835.514,-260.423,-544.761,-89.9199,-0.9682,180.0004
C03136=1980.580,-260.409,-544.761,-92.5040,-0.7391,-179.9660
C03137=1848.362,-260.392,-544.761,-91.4841,-0.8021,-179.9775
C03138=1831.829,-260.365,-544.761,-89.7309,-2.8819,179.9889
C03139=2135.648,-260.354,-544.761,-91.4039,0.5844,179.9832
C03140=1920.149,-260.334,-544.761,-92.1373,0.2521,179.9889
C03141=1873.512,-260.317,-544.761,-91.0831,-0.5156,-179.9889
C03142=2090.011,-260.305,-544.761,-92.0972,0.2578,179.9889
C03143=1999.619,-260.288,-544.761,-91.5013,-0.0974,-179.9946
C03144=2118.771,-260.267,-544.761,-91.2320,0.7906,179.9832
C03145=1893.437,-260.253,-544.761,-91.5987,-0.3036,-179.9889
C03146=1995.325,-260.237,-544.761,-92.6358,-0.2062,-179.9889
C03147=1877.827,-260.217,-544.761,-91.3638,-1.1115,-179.9717
C03148=1861.590,-260.198,-544.761,-92.1144,-0.5614,-179.9775
C03149=1949.022,-260.188,-544.761,-91.9310,0.0458,180.0004
C03150=2065.874,-260.160,-544.761,-92.1889,0.2234,179.9889
C03151=1984.529,-260.117,-544.761,-91.6388,-0.4182,-179.9889
C03152=1946.014,-260.067,-544.761,-91.9196,-0.0859,-179.9946
C03153=2028.490,-260.046,-544.761,-90.9455,1.4610,179.9775
C03154=1878.387,-260.014,-544.761,-91.4956,-1.1344,-179.9717
C03155=2054.593,-260.005,-544.761,-92.7504,-0.3323,-179.9832
C03156=2072.406,-259.984,-544.761,-92.4295,-0.0229,-180.0004
C03157=1954.819,-259.971,-544.761,-92.7675,-0.3495,-179.9832
C03158=2079.669,-259.920,-544.761,-92.1488,0.1203,179.9946
C03159=2034.819,-259.900,-544.761,-92.8306,0.3265,179.9832
C03160=2001.013,-259.884,-544.761,-90.7278,0.5042,179.9946
C03161=1936.039,-259.870,-544.761,-92.4123,-0.3896,-179.9832
C03162=2016.505,-259.830,-544.761,-91.4612,-1.3292,-179.9660
C03163=2105.713,-259.797,-544.761,-92.2920,0.6818,179.9717
C03164=1928.160,-259.790,-544.761,-92.3378,0.5213,179.9775
C03165=2100.667,-259.760,-544.761,-92.5899,0.3380,179.9832
C03166=1968.585,-259.715,-544.761,-92.5498,1.9194,179.9144
C03167=1957.890,-259.692,-544.761,-92.4467,1.1115,179.9545
C03168=1907.944,-259.650,-544.761,-92.4123,-0.9281,-179.9603
C03169=2022.531,-259.635,-544.761,-91.6445,-0.2692,-179.9946
C03170=2045.046,-259.595,-544.761,-91.8795,-0.8823,-179.9717
C03171=1945.854,-259.558,-544.761,-93.8161,0.6187,179.9603
C03172=2035.480,-259.537,-544.761,-92.2290,0.8078,179.9660
C03173=2051.644,-259.510,-544.761,-92.5040,-0.7849,-179.9660
C03174=2087.205,-259.470,-544.761,-91.2320,0.3495,179.9946
C03175=1976.162,-259.450,-544.761,-93.3749,0.4812,179.9717
C03176=1946.439,-259.404,-544.761,-91.6732,-0.1145,-179.9946
C03177=1957.313,-259.374,-544.761,-92.0284,-0.4984,-179.9832
C03178=2083.156,-259.348,-544.761,-90.7622,-0.0401,-180.0004
C03179=1979.022,-259.233,-544.761,-90.7221,-0.1203,-180.0004
C03180=1975.506,-257.856,-594.761,-92.1086,-0.3896,-179.9832
C03181=2006.601,-257.960,-594.761,-91.5529,0.8193,179.9775
C03182=2043.583,-257.974,-594.761,-90.7966,0.0000,180.0004
C03183=2076.505,-257.997,-594.761,-91.1919,0.5729,179.9889
C03184=2005.853,-258.029,-594.761,-91.9998,0.1776,179.9946
C03185=1968.632,-258.047,-594.761,-91.0200,0.1489,179.9946
C03186=1950.789,-258.061,-594.761,-91.6503,-0.1718,-179.9946
C03187=1936.259,-258.086,-594.761,-91.1174,0.6990,179.9889
C03188=1945.613,-258.125,-594.761,-91.9597,-1.8048,-179.9373
C03189=2075.447,-258.155,-594.761,-91.1232,-0.0802,-180.0004
C03190=1950.546,-258.173,-594.761,-92.3837,-0.6646,-179.9717
C03191=1926.315,-258.193,-594.761,-90.7679,-0.3838,-179.9946
C03192=1982.653,-258.200,-594.761,-90.5960,0.7391,179.9946
C03193=1978.382,-258.235,-594.761,-91.9597,-0.1031,-179.9946
C03194=2019.060,-258.261,-594.761,-91.5471,-0.1031,-179.9946
C03195=1947.702,-258.288,-594.761,-91.2950,-0.0343,-180.0004
C03196=2010.528,-258.308,-594.761,-90.6361,-0.5901,-179.9946
C03197=1974.208,-258.315,-594.761,-91.3867,-0.2463,-179.9946
C03198=2047.057,-258.336,-594.761,-90.7565,0.7104,179.9889
C03199=2110.855,-258.380,-594.761,-90.5330,1.3636,179.9889
C03200=1897.268,-258.412,-594.761,-91.0773,0.8479,179.9832
C03201=1934.923,-258.446,-594.761,-90.9284,-0.2119,-179.9946
C03202=2062.708,-258.475,-594.761,-92.8764,-1.0084,-179.9488
C03203=1991.921,-258.489,-594.761,-90.9914,-0.0401,-180.0004
C03204=2071.862,-258.515,-594.761,-91.4383,0.0572,180.0004
C03205=2077.376,-258.534,-594.761,-92.0685,0.8594,179.9717
C03206=1885.348,-258.538,-594.761,-89.7022,0.1317,-180.0004
C03207=1982.583,-258.548,-594.761,-91.4784,-0.5844,-179.9832
C03208=1900.176,-258.564,-594.761,-91.2893,-0.0687,-180.0004
C03209=1966.706,-258.589,-594.761,-90.8138,0.7620,179.9889
C03210=2107.198,-258.596,-594.761,-90.9971,0.4583,179.9946
C03211=2059.464,-258.620,-594.761,-91.3409,-0.1031,-180.0004
C03212=1910.029,-258.641,-594.761,-91.4326,-0.4469,-179.9889
C03213=2118.898,-258.685,-594.761,-90.8539,1.2891,179.9832
C03214=1883.168,-258.709,-594.761,-91.0601,-0.7563,-179.9832
C03215=2032.730,-258.733,-594.761,-91.8909,0.3380,179.9889
C03216=2039.315,-258.747,-594.761,-92.2175,0.0114,180.0004
C03217=1906.954,-258.789,-594.761,-92.3149,0.1890,179.9946
C03218=2122.856,-258.799,-594.761,-90.3325,1.5699,179.9889
C03219=1937.499,-258.819,-594.761,-91.7420,0.4297,179.9889
C03220=2076.275,-258.844,-594.761,-91.7992,0.6073,179.9832
C03221=2006.823,-258.871,-594.761,-90.8768,0.2234,179.9946
C03222=1892.551,-258.879,-594.761,-91.3982,-0.6875,-179.9832
C03223=2014.743,-258.919,-594.761,-91.3695,0.5844,179.9832
C03224=2074.409,-258.971,-594.761,-92.5212,0.3552,179.9832
C03225=1921.246,-258.981,-594.761,-91.4956,0.0458,180.0004
C03226=2056.623,-259.012,-594.761,-92.3092,0.7906,179.9660
C03227=1976.930,-259.023,-594.761,-91.0601,-0.3265,-179.9946
C03228=1888.774,-259.039,-594.761,-91.1976,-1.0026,-179.9775
C03229=1875.304,-259.056,-594.761,-91.7076,-0.2234,-179.9946
C03230=1907.160,-259.075,-594.761,-92.2863,0.0171,180.0004
C03231=1887.079,-259.105,-594.761,-90.7622,-1.2433,-179.9832
C03232=1936.288,-259.118,-594.761,-92.4352,0.3838,179.9832
C03233=2040.977,-259.134,-594.761,-90.9455,-0.3437,-179.9946
C03234=2128.164,-259.163,-594.761,-91.3982,1.3006,179.9660
C03235=2072.801,-259.188,-594.761,-92.1373,0.4297,179.9832
C03236=1871.532,-259.218,-594.761,-90.7679,-1.9881,-179.9717
C03237=2034.112,-259.246,-594.761,-91.9941,-0.1317,-179.9946
C03238=1862.458,-259.269,-594.761,-91.5873,-1.4037,-179.9603
C03239=1857.782,-259.295,-594.761,-91.0487,-1.7647,-179.9660
C03240=1964.076,-259.322,-594.761,-92.1029,0.7677,179.9717
C03241=2047.145,-259.352,-594.761,-92.8535,-1.3865,-179.9316
C03242=1880.959,-259.406,-594.761,-91.4268,-0.7964,-179.9775
C03243=2004.925,-259.456,-594.761,-91.5987,0.9281,179.9717
C03244=2099.609,-259.488,-594.761,-91.7763,2.0511,179.9373
C03245=2144.537,-259.524,-594.761,-90.8424,2.3548,179.9660
C03246=2105.933,-259.586,-594.761,-92.0399,0.5958,179.9775
C03247=1848.169,-259.648,-594.761,-90.0746,-1.8735,-180.0004
C03248=1847.758,-259.734,-594.761,-90.5502,-1.6100,-179.9832
C03249=2144.235,-259.767,-594.761,-91.5185,2.5152,179.9316
C03250=1842.596,-259.859,-594.761,-90.7966,-1.3750,-179.9832
C03251=2136.079,-259.888,-594.761,-91.5300,1.5756,179.9603
C03252=2143.069,-259.985,-594.761,-91.5815,1.5412,179.9603
C03253=1840.442,-260.007,-594.761,-90.0746,-2.3433,-179.9946
C03254=1836.528,-260.061,-594.761,-90.3898,-2.0110,-179.9889
C03255=2161.067,-260.162,-594.761,-89.9486,3.2773,-179.9946
C03256=1833.421,-260.234,-594.761,-90.3497,-2.7616,-179.9832
C03257=2156.691,-260.301,-594.761,-91.3180,1.9194,179.9545
C03258=1828.131,-260.435,-594.761,-90.4872,0.3437,179.9946
C03259=1822.949,-260.521,-594.761,-90.4012,-2.3204,-179.9832
C03260=2169.354,-260.567,-594.761,-90.0002,2.9450,180.0004
C03261=1820.066,-260.698,-594.761,-89.7710,-1.8735,179.9946
C03262=1821.878,-260.763,-594.761,-90.1549,-2.4522,-179.9946
C03263=1815.778,-260.860,-594.761,-89.2954,-1.9136,179.9775
C03264=2176.814,-260.934,-594.761,-90.6763,3.2544,179.9603
C03265=2172.570,-260.978,-594.761,-90.5674,2.2746,179.9775
C03266=1809.014,-261.035,-594.761,-90.0059,-2.0626,-180.0004
C03267=1812.378,-261.091,-594.761,-89.9944,-2.4866,180.0004
C03268=1811.469,-261.134,-594.761,-89.5876,-3.0309,179.9775
C03269=1806.242,-261.193,-594.761,-89.1293,-2.3548,179.9660
C03270=1799.144,-261.309,-594.761,-88.9918,-3.2887,179.9431
C03271=1796.063,-261.353,-594.761,-88.1266,7.4656,-179.7540
C03272=1800.022,-261.367,-594.761,-88.9001,-1.7647,179.9660
C03273=1802.737,-261.531,-594.761,-89.3814,-3.0653,179.9660
C03274=1795.613,-261.580,-594.761,-87.2156,0.6531,-179.9660
C03275=2187.688,-261.652,-594.761,-89.8569,3.4320,-179.9889
C03276=1797.468,-261.768,-594.761,-88.8772,-2.8762,179.9431
C03277=2190.839,-261.875,-594.761,-91.0315,1.5355,179.9717
C03278=1797.016,-261.995,-594.761,-88.8600,2.8934,-179.9431
C03279=1798.970,-262.465,-644.761,-88.8141,-2.6929,179.9431
C03280=1796.247,-262.211,-644.761,-89.5475,-0.4010,179.9946
C03281=2191.211,-262.002,-644.761,-87.5364,-0.0802,179.9946
C03282=1803.707,-261.891,-644.761,-89.6793,-5.9931,179.9660
C03283=1803.478,-261.793,-644.761,-89.3986,-3.2773,179.9660
C03284=2187.072,-261.722,-644.761,-88.8256,4.1825,-179.9144
C03285=2193.651,-261.661,-644.761,-91.9769,-13.6765,-179.5305
C03286=2187.221,-261.583,-644.761,-89.7137,3.4606,-179.9832
C03287=1804.257,-261.440,-644.761,-90.5445,-4.5722,-179.9545
C03288=1811.483,-261.369,-644.761,-89.0777,-3.9820,179.9373
C03289=1810.682,-261.260,-644.761,-90.7794,-2.9335,-179.9603
C03290=2177.467,-261.107,-644.761,-90.1549,3.8273,179.9889
C03291=2177.509,-260.994,-644.761,-89.7022,3.1799,-179.9832
C03292=1821.215,-260.865,-644.761,-90.0976,-2.9278,-179.9946
C03293=2172.041,-260.749,-644.761,-89.7423,3.1054,-179.9889
C03294=2170.868,-260.702,-644.761,-90.2866,3.0939,179.9832
C03295=1828.065,-260.492,-644.761,-91.1633,-3.0080,-179.9373
C03296=1832.099,-260.313,-644.761,-90.4241,-3.2257,-179.9775
C03297=2164.047,-260.166,-644.761,-88.7511,2.7960,-179.9373
C03298=1836.783,-260.034,-644.761,-89.6277,-2.5897,179.9832
C03299=2156.915,-259.932,-644.761,-89.7595,2.6356,-179.9889
C03300=1842.827,-259.797,-644.761,-90.1491,-3.1684,-179.9889
C03301=1836.341,-259.756,-644.761,-91.3237,-1.7761,-179.9603
C03302=1845.845,-259.557,-644.761,-89.3928,-3.9705,179.9603
C03303=1850.073,-259.457,-644.761,-90.2866,-2.6413,-179.9889
C03304=1853.851,-259.396,-644.761,-90.6247,-1.9423,-179.9775
C03305=1847.099,-259.295,-644.761,-89.0777,-2.8705,179.9545
C03306=2141.896,-259.242,-644.761,-89.6736,2.8246,-179.9832
C03307=1856.964,-259.117,-644.761,-90.2752,-2.2173,-179.9889
C03308=1861.627,-259.005,-644.761,-89.2439,-2.5954,179.9660
C03309=1859.827,-258.931,-644.761,-90.5101,-2.1715,-179.9832
C03310=1871.831,-258.822,-644.761,-90.0575,-1.7647,-180.0004
C03311=1865.678,-258.764,-644.761,-89.4272,-1.5985,179.9832
C03312=2122.715,-258.728,-644.761,-91.0086,1.3636,179.9775
C03313=2117.886,-258.659,-644.761,-89.5246,2.0340,-179.9832
C03314=1871.010,-258.626,-644.761,-90.2924,-2.3835,-179.9889
C03315=1876.193,-258.563,-644.761,-91.4211,-1.7188,-179.9545
C03316=2116.714,-258.509,-644.761,-91.2091,0.6417,179.9889
C03317=1885.146,-258.430,-644.761,-91.9883,-1.8850,-179.9373
C03318=2114.671,-258.362,-644.761,-90.1892,1.3865,179.9946
C03319=1872.610,-258.298,-644.761,-90.8481,-1.7016,-179.9775
C03320=1882.136,-258.248,-644.761,-89.5590,-1.8220,179.9832
C03321=1895.852,-258.212,-644.761,-90.1663,-1.4438,-179.9946
C03322=1889.422,-258.161,-644.761,-90.9169,-1.0657,-179.9832
C03323=2102.364,-258.132,-644.761,-89.8397,0.7734,-180.0004
C03324=2101.942,-258.108,-644.761,-90.1262,0.8995,180.0004
C03325=1899.936,-258.068,-644.761,-90.4070,-1.0828,-179.9946
C03326=2103.695,-258.025,-644.761,-89.7882,1.1401,-179.9946
C03327=2082.194,-257.993,-644.761,-91.2091,1.4438,179.9717
C03328=2076.015,-257.952,-644.761,-90.5158,0.7276,179.9946
C03329=1910.703,-257.931,-644.761,-91.0601,-0.4526,-179.9889
C03330=1917.100,-257.917,-644.761,-90.7851,-0.3896,-179.9946
C03331=1940.719,-257.905,-644.761,-91.3065,-0.2692,-179.9946
C03332=1961.928,-257.889,-644.761,-91.1461,0.2635,179.9946
C03333=2090.408,-257.871,-644.761,-90.5846,0.9396,179.9889
C03334=2072.946,-257.854,-644.761,-90.3840,1.3407,179.9889
C03335=1910.699,-257.840,-644.761,-88.9230,0.9052,-179.9832
C03336=2023.164,-257.823,-644.761,-91.0028,-0.0171,-180.0004
C03337=2084.155,-257.804,-644.761,-90.8138,0.3437,179.9946
C03338=2012.223,-257.788,-644.761,-91.5930,-0.0343,-180.0004
C03339=1936.512,-257.780,-644.761,-90.6705,-0.2234,-179.9946
C03340=1919.876,-257.759,-644.761,-90.7507,-0.8537,-179.9889
C03341=2002.111,-257.748,-644.761,-90.2465,-0.6646,-179.9946
C03342=2018.400,-257.732,-644.761,-91.1232,0.5156,179.9889
C03343=2064.837,-257.722,-644.761,-89.7939,0.5500,-180.0004
C03344=2081.925,-257.710,-644.761,-89.5189,0.3666,-179.9946
C03345=2037.211,-257.700,-644.761,-90.4299,-0.9167,-179.9946
C03346=1993.727,-257.689,-644.761,-91.4268,-0.1031,-179.9946
C03347=2001.922,-257.685,-644.761,-90.9971,0.4125,179.9946
C03348=1930.788,-257.678,-644.761,-91.2893,-0.5213,-179.9889
C03349=1900.989,-257.669,-644.761,-91.4497,-0.7964,-179.9775
C03350=1937.710,-257.660,-644.761,-90.6820,-0.4182,-179.9946
C03351=2083.356,-257.652,-644.761,-90.2523,0.4182,180.0004
C03352=1967.410,-257.646,-644.761,-91.1690,-0.2979,-179.9946
C03353=1925.347,-257.641,-644.761,-90.5387,-0.8250,-179.9946
C03354=1958.648,-257.624,-644.761,-91.0086,0.2406,179.9946
C03355=2037.434,-257.617,-644.761,-91.2549,-0.0802,-180.0004
C03356=1899.387,-257.605,-644.761,-90.5044,-1.3464,-179.9889
C03357=2025.422,-257.589,-644.761,-92.0112,0.5271,179.9832
C03358=1975.027,-257.575,-644.761,-91.9138,1.8220,179.9373
C03359=1915.038,-257.549,-644.761,-90.3497,-0.6760,-179.9946
C03360=1972.643,-257.539,-644.761,-91.0315,0.7505,179.9889
C03361=1959.202,-257.523,-644.761,-91.0315,1.2204,179.9775
C03362=1951.110,-257.510,-644.761,-90.2122,-0.0114,-180.0004
C03363=2010.252,-257.502,-644.761,-89.3928,-0.5156,179.9946
C03364=1928.495,-257.494,-644.761,-91.0888,0.3781,179.9946
C03365=2029.678,-257.485,-644.761,-91.0945,-0.4526,-179.9889
C03366=1953.653,-257.474,-644.761,-90.0575,-0.3208,-180.0004
C03367=1941.790,-257.458,-644.761,-90.4127,-0.0171,-180.0004
C03368=2020.357,-257.444,-644.761,-90.2465,0.3896,180.0004
C03369=2043.800,-257.430,-644.761,-89.5475,-1.1229,179.9889
C03370=1953.336,-257.408,-644.761,-91.0372,0.0802,180.0004
C03371=1974.292,-257.387,-644.761,-89.9658,0.1203,-180.0004
C03372=1965.413,-257.369,-644.761,-90.4700,-1.0255,-179.9889
C03373=2005.907,-257.337,-644.761,-91.2950,-0.5557,-179.9889
C03374=1967.602,-257.314,-644.761,-90.2007,-0.1031,-180.0004
C03375=1947.102,-257.138,-694.761,-90.8711,0.3323,179.9946
C03376=1999.192,-257.207,-694.761,-90.4757,0.3208,179.9946
C03377=1948.866,-257.230,-694.761,-89.2668,0.0802,-180.0004
C03378=1942.446,-257.262,-694.761,-89.8283,-0.3036,180.0004
C03379=1955.709,-257.274,-694.761,-89.7481,0.3437,-180.0004
C03380=2008.496,-257.286,-694.761,-90.1491,-0.0630,-180.0004
C03381=1985.093,-257.298,-694.761,-89.7710,-0.0343,180.0004
C03382=1921.908,-257.314,-694.761,-89.7481,0.1718,-180.0004
C03383=1933.695,-257.326,-694.761,-89.6736,-0.6474,179.9946
C03384=1928.511,-257.341,-694.761,-89.7137,-0.1317,180.0004
C03385=2015.374,-257.357,-694.761,-89.7423,-0.0343,180.0004
C03386=1972.311,-257.364,-694.761,-89.8798,0.0229,-180.0004
C03387=2013.357,-257.370,-694.761,-90.4070,0.1546,180.0004
C03388=1942.638,-257.379,-694.761,-89.2381,0.1088,-180.0004
C03389=2030.388,-257.394,-694.761,-89.3699,0.2119,-180.0004
C03390=2023.263,-257.401,-694.761,-88.5448,0.2062,-179.9946
C03391=1993.455,-257.407,-694.761,-90.2580,0.3495,180.0004
C03392=1914.113,-257.412,-694.761,-89.8111,-0.7391,179.9946
C03393=1957.645,-257.418,-694.761,-88.6365,0.0286,-180.0004
C03394=1915.229,-257.423,-694.761,-89.6793,-0.3323,180.0004
C03395=2035.118,-257.430,-694.761,-90.1606,1.3063,179.9946
C03396=2042.432,-257.437,-694.761,-89.7882,-1.1344,179.9946
C03397=1960.369,-257.459,-694.761,-89.7882,0.3552,-180.0004
C03398=1912.767,-257.480,-694.761,-90.4127,-0.1604,-180.0004
C03399=1920.555,-257.490,-694.761,-90.2408,-0.0687,-180.0004
C03400=2049.461,-257.496,-694.761,-89.5189,0.7906,-179.9946
C03401=1909.195,-257.516,-694.761,-89.8111,-0.2062,180.0004
C03402=2035.464,-257.533,-694.761,-89.5991,0.4354,-179.9946
C03403=1905.283,-257.545,-694.761,-90.7679,-0.7563,-179.9889
C03404=2030.623,-257.556,-694.761,-88.9803,-0.5443,179.9889
C03405=1890.242,-257.577,-694.761,-90.3497,-0.9224,-179.9946
C03406=2025.437,-257.603,-694.761,-88.9402,1.1000,-179.9775
C03407=2041.125,-257.627,-694.761,-89.6793,-1.3980,179.9946
C03408=1984.875,-257.644,-694.761,-89.0032,0.2349,-179.9946
C03409=1898.180,-257.657,-694.761,-90.3382,0.0171,180.0004
C03410=2066.220,-257.669,-694.761,-89.6793,0.2578,-180.0004
C03411=2074.116,-257.694,-694.761,-89.7595,0.5901,-179.9946
C03412=1888.206,-257.725,-694.761,-90.9570,-1.6902,-179.9717
C03413=2062.616,-257.755,-694.761,-89.2897,0.1661,-180.0004
C03414=2045.907,-257.785,-694.761,-89.2725,0.5557,-179.9946
C03415=1889.336,-257.813,-694.761,-90.0517,-1.6730,-180.0004
C03416=2031.982,-257.833,-694.761,-89.3584,-0.2291,179.9946
C03417=2052.273,-257.864,-694.761,-88.9459,0.9453,-179.9832
C03418=2083.032,-257.899,-694.761,-89.1006,1.1344,-179.9832
C03419=2092.348,-257.944,-694.761,-89.2610,1.3292,-179.9832
C03420=1884.475,-257.982,-694.761,-91.4211,-1.2662,-179.9660
C03421=1869.344,-258.030,-694.761,-90.2408,-1.7131,-179.9946
C03422=1868.652,-258.054,-694.761,-92.0743,-0.0630,-180.0004
C03423=2058.761,-258.080,-694.761,-88.8371,1.2834,-179.9717
C03424=1862.957,-258.152,-694.761,-90.0002,-1.3980,180.0004
C03425=2090.167,-258.202,-694.761,-88.7511,0.9052,-179.9775
C03426=2069.807,-258.251,-694.761,-88.7511,0.4526,-179.9889
C03427=1870.433,-258.324,-694.761,-90.6190,-1.0714,-179.9889
C03428=2089.421,-258.392,-694.761,-88.7110,0.8307,-179.9832
C03429=2096.217,-258.445,-694.761,-89.0605,1.3980,-179.9775
C03430=1850.421,-258.527,-694.761,-90.0632,-2.1199,-180.0004
C03431=1851.975,-258.646,-694.761,-90.8596,-2.6527,-179.9603
C03432=2120.879,-258.712,-694.761,-89.7481,-0.0687,180.0004
C03433=1846.345,-258.807,-694.761,-90.2981,-1.8964,-179.9889
C03434=1843.146,-258.826,-694.761,-90.7507,-2.0798,-179.9717
C03435=1845.750,-258.936,-694.761,-91.0258,-2.2402,-179.9603
C03436=2128.259,-259.010,-694.761,-89.6850,1.9194,-179.9889
C03437=1833.874,-259.039,-694.761,-90.9856,-2.8418,-179.9488
C03438=2133.807,-259.216,-694.761,-89.2897,1.9709,-179.9775
C03439=1838.098,-259.285,-694.761,-90.8768,-2.3605,-179.9660
C03440=2117.638,-259.365,-694.761,-88.6365,1.6329,-179.9603
C03441=2123.799,-259.451,-694.761,-88.4589,1.9365,-179.9488
C03442=2135.773,-259.596,-694.761,-88.3730,1.9595,-179.9431
C03443=1821.995,-259.699,-694.761,-91.3523,-3.0252,-179.9259
C03444=1827.408,-259.856,-694.761,-90.9742,-2.7100,-179.9545
C03445=2146.457,-259.907,-694.761,-88.2756,2.4350,-179.9259
C03446=1817.310,-260.023,-694.761,-90.9226,-2.5897,-179.9603
C03447=1816.417,-260.092,-694.761,-90.9799,-2.8590,-179.9488
C03448=1829.021,-260.137,-694.761,-91.7133,-2.7158,-179.9202
C03449=1812.424,-260.433,-694.761,-91.6617,-2.7387,-179.9202
C03450=1805.310,-260.506,-694.761,-90.8825,-2.6184,-179.9603
C03451=2155.195,-260.532,-694.761,-89.1636,2.8934,-179.9603
C03452=1801.471,-260.674,-694.761,-91.7362,-2.8762,-179.9144
C03453=2161.924,-260.829,-694.761,-88.7683,1.8964,-179.9603
C03454=2173.333,-260.918,-694.761,-88.7912,3.6955,-179.9202
C03455=1793.567,-261.027,-694.761,-93.3520,18.8675,178.9175
C03456=1798.268,-261.151,-694.761,-91.5013,-2.8877,-179.9259
C03457=2177.388,-261.248,-694.761,-89.5762,3.0538,-179.9775
C03458=2174.096,-261.393,-694.761,-88.9688,3.0424,-179.9431
C03459=1805.813,-261.482,-694.761,-90.7737,-3.7070,-179.9488
C03460=1795.196,-261.623,-694.761,-89.8970,6.5546,-179.9889
C03461=1793.535,-261.809,-694.761,-92.0800,8.5485,179.6910
C03462=2183.607,-261.944,-694.761,-89.2668,3.3174,-179.9603
C03463=2186.836,-262.175,-694.761,-88.6766,3.8216,-179.9144
C03464=2191.049,-262.383,-694.761,-88.7053,-2.4006,179.9431
C03465=2192.205,-262.721,-744.761,-89.2725,-9.2303,179.8858
C03466=2186.150,-262.552,-744.761,-89.5762,2.0626,-179.9832
C03467=2181.639,-262.451,-744.761,-89.1636,2.1142,-179.9717
C03468=2188.040,-262.361,-744.761,-90.4643,2.1543,179.9832
C03469=2193.286,-262.254,-744.761,-90.7278,-16.0141,-179.7998
C03470=2169.038,-262.158,-744.761,-89.1751,1.1516,-179.9832
C03471=2174.293,-262.023,-744.761,-89.1866,1.9308,-179.9717
C03472=2165.569,-261.801,-744.761,-89.1293,1.7532,-179.9717
C03473=2172.003,-261.704,-744.761,-88.7626,2.6699,-179.9431
C03474=2147.913,-261.463,-744.761,-88.5563,1.5011,-179.9603
C03475=2168.241,-261.324,-744.761,-88.7855,2.7158,-179.9431
